KUKA KRL program: MyProgram_319().src

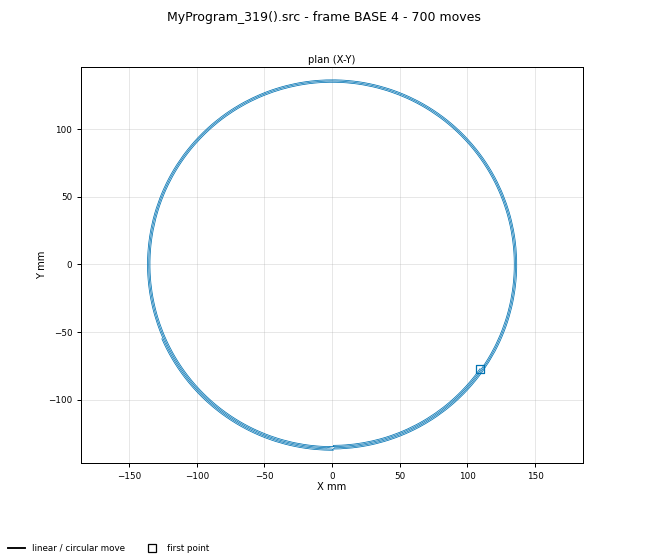
[picture p0: tool path of MyProgram_319().src in frame BASE 4, 700 of 700 moves have a stored position in this frame; points joined in program order, loops and branches not executed]
&ACCESS RVP
&REL 1
&PARAM TEMPLATE = C:\KRC\Roboter\Template\vorgabe
&PARAM EDITMASK = *
DEF MyProgram_319()
; ---- Setting reference (Base) ----
$BASE = BASE_DATA[4]

; --------------------------
; ---- Setting tool (TCP) ----
$TOOL = TOOL_DATA[3]
; --------------------------

$VEL.CP = VEL_APROX_PRINT
Startdeposition()
$VEL.CP = VEL_PRINT
LIN {X 109.3778,Y -77.0106,Z 185,A -30.8894,B 3.0839,C 0.2483,E1 3.2253,E2 483.8317} C_DIS
LIN {X 107.5202,Y -79.5843,Z 185,A -32.1533,B 3.0837,C 0.2506,E1 3.2233,E2 485.0845} C_DIS
LIN {X 105.6235,Y -82.0842,Z 185,A -33.5327,B 3.0834,C 0.2541,E1 3.2209,E2 486.4695} C_DIS
LIN {X 103.4321,Y -84.829,Z 185,A -34.958,B 3.0832,C 0.2567,E1 3.2184,E2 487.886} C_DIS
LIN {X 100.7853,Y -87.957,Z 185,A -36.6496,B 3.0829,C 0.26,E1 3.2154,E2 489.5709} C_DIS
LIN {X 98.5631,Y -90.4402,Z 185,A -38.0166,B 3.0827,C 0.2625,E1 3.2128,E2 490.9313} C_DIS
LIN {X 95.7665,Y -93.3971,Z 185,A -39.7017,B 3.0825,C 0.2657,E1 3.2096,E2 492.6104} C_DIS
LIN {X 93.4185,Y -95.7456,Z 185,A -41.0913,B 3.0822,C 0.2683,E1 3.2068,E2 493.997} C_DIS
LIN {X 90.4442,Y -98.5594,Z 185,A -42.9213,B 3.0819,C 0.2726,E1 3.203,E2 495.8381} C_DIS
LIN {X 87.3741,Y -101.2911,Z 185,A -44.4719,B 3.0817,C 0.2741,E1 3.1998,E2 497.3634} C_DIS
LIN {X 84.3456,Y -103.8272,Z 185,A -46.1519,B 3.0814,C 0.2772,E1 3.1962,E2 499.0432} C_DIS
LIN {X 81.6511,Y -105.9592,Z 185,A -47.6942,B 3.0811,C 0.2805,E1 3.1928,E2 500.5957} C_DIS
LIN {X 78.452,Y -108.3485,Z 185,A -49.2173,B 3.0811,C 0.2819,E1 3.1894,E2 502.0961} C_DIS
LIN {X 76.0517,Y -110.0474,Z 185,A -50.5208,B 3.0808,C 0.2845,E1 3.1864,E2 503.4062} C_DIS
LIN {X 72.8711,Y -112.1781,Z 185,A -52.0108,B 3.0807,C 0.2859,E1 3.183,E2 504.8783} C_DIS
LIN {X 70.2032,Y -113.8671,Z 185,A -53.3655,B 3.0804,C 0.2881,E1 3.1798,E2 506.2343} C_DIS
LIN {X 67.5529,Y -115.459,Z 185,A -54.6759,B 3.0803,C 0.2901,E1 3.1766,E2 507.5439} C_DIS
LIN {X 64.5814,Y -117.147,Z 185,A -56.059,B 3.0801,C 0.2916,E1 3.1733,E2 508.9177} C_DIS
LIN {X 61.6787,Y -118.6998,Z 185,A -57.4546,B 3.0799,C 0.2935,E1 3.1698,E2 510.3125} C_DIS
LIN {X 58.6673,Y -120.2166,Z 185,A -58.8657,B 3.0798,C 0.2952,E1 3.1663,E2 511.7203} C_DIS
LIN {X 55.7023,Y -121.6185,Z 185,A -60.239,B 3.0796,C 0.2968,E1 3.1628,E2 513.0906} C_DIS
LIN {X 53.1765,Y -122.743,Z 185,A -61.4788,B 3.0794,C 0.2988,E1 3.1596,E2 514.3383} C_DIS
LIN {X 49.6723,Y -124.203,Z 185,A -62.991,B 3.0794,C 0.2998,E1 3.1558,E2 515.837} C_DIS
LIN {X 46.6127,Y -125.3832,Z 185,A -64.3692,B 3.0792,C 0.3012,E1 3.1522,E2 517.2128} C_DIS
LIN {X 43.5231,Y -126.4889,Z 185,A -65.8758,B 3.079,C 0.3035,E1 3.1481,E2 518.7333} C_DIS
LIN {X 39.4666,Y -127.8128,Z 185,A -67.6587,B 3.0788,C 0.305,E1 3.1434,E2 520.5116} C_DIS
LIN {X 35.6745,Y -128.9228,Z 185,A -69.2121,B 3.0788,C 0.3055,E1 3.1393,E2 522.0482} C_DIS
LIN {X 32.5911,Y -129.7365,Z 185,A -70.5581,B 3.0787,C 0.3065,E1 3.1356,E2 523.3925} C_DIS
LIN {X 29.3997,Y -130.497,Z 185,A -71.9433,B 3.0786,C 0.3075,E1 3.1319,E2 524.776} C_DIS
LIN {X 26.191,Y -131.179,Z 185,A -73.3307,B 3.0785,C 0.3084,E1 3.1281,E2 526.162} C_DIS
LIN {X 22.9498,Y -131.7853,Z 185,A -74.7231,B 3.0785,C 0.3091,E1 3.1242,E2 527.5527} C_DIS
LIN {X 19.6218,Y -132.3222,Z 185,A -76.1756,B 3.0783,C 0.3101,E1 3.1202,E2 529.0071} C_DIS
LIN {X 16.4658,Y -132.7515,Z 185,A -77.5281,B 3.0783,C 0.3107,E1 3.1165,E2 530.3588} C_DIS
LIN {X 13.2073,Y -133.1144,Z 185,A -78.924,B 3.0782,C 0.3113,E1 3.1126,E2 531.7544} C_DIS
LIN {X 9.919,Y -133.3992,Z 185,A -80.3167,B 3.0782,C 0.3117,E1 3.1087,E2 533.1452} C_DIS
LIN {X 6.649,Y -133.6021,Z 185,A -81.7182,B 3.0782,C 0.3121,E1 3.1048,E2 534.5471} C_DIS
LIN {X 3.2803,Y -133.7279,Z 185,A -83.13,B 3.0781,C 0.3123,E1 3.1009,E2 535.9555} C_DIS
LIN {X 0.9683,Y -133.7631,Z 185,A -83.8532,B 3.0783,C 0.3106,E1 3.0989,E2 536.6446} C_DIS
Enddeposition()
LIN {X 0.9683,Y -133.7631,Z 185,A -83.8532,B 3.0783,C 0.3106,E1 3.0989,E2 536.6446} C_DIS
Startdeposition()
$VEL.CP = VEL_PRINT
LIN {X 1.3005,Y -134.6625,Z 185,A -83.2219,B 3.0781,C 0.3087,E1 3.1005,E2 535.98} C_DIS
LIN {X 4.845,Y -134.581,Z 185,A -81.7788,B 3.0781,C 0.3087,E1 3.1045,E2 534.5448} C_DIS
LIN {X 8.4966,Y -134.3994,Z 185,A -79.9996,B 3.0784,C 0.3065,E1 3.1095,E2 532.7353} C_DIS
LIN {X 11.7944,Y -134.1508,Z 185,A -78.8459,B 3.0782,C 0.3079,E1 3.1127,E2 531.6142} C_DIS
LIN {X 15.0407,Y -133.8264,Z 185,A -77.5552,B 3.0782,C 0.3079,E1 3.1162,E2 530.3356} C_DIS
LIN {X 18.6503,Y -133.3703,Z 185,A -76.1047,B 3.0782,C 0.3079,E1 3.1202,E2 528.897} C_DIS
LIN {X 22.1894,Y -132.8267,Z 185,A -74.5857,B 3.0783,C 0.307,E1 3.1244,E2 527.3777} C_DIS
LIN {X 26.0809,Y -132.12,Z 185,A -72.6662,B 3.0786,C 0.304,E1 3.1298,E2 525.4261} C_DIS
LIN {X 29.5428,Y -131.3876,Z 185,A -71.3256,B 3.0786,C 0.3042,E1 3.1334,E2 524.1063} C_DIS
LIN {X 32.2356,Y -130.7541,Z 185,A -70.0345,B 3.0788,C 0.3023,E1 3.1369,E2 522.7994} C_DIS
LIN {X 36.5633,Y -129.6089,Z 185,A -68.2253,B 3.0788,C 0.3013,E1 3.1418,E2 521.0015} C_DIS
LIN {X 40.7406,Y -128.357,Z 185,A -66.4521,B 3.079,C 0.3002,E1 3.1465,E2 519.238} C_DIS
LIN {X 44.2028,Y -127.206,Z 185,A -64.9326,B 3.0791,C 0.2988,E1 3.1505,E2 517.7217} C_DIS
LIN {X 46.9299,Y -126.2257,Z 185,A -63.7404,B 3.0792,C 0.2978,E1 3.1536,E2 516.534} C_DIS
LIN {X 50.2109,Y -124.9564,Z 185,A -62.2458,B 3.0794,C 0.296,E1 3.1575,E2 515.0386} C_DIS
LIN {X 53.1011,Y -123.7563,Z 185,A -61.1043,B 3.0794,C 0.296,E1 3.1604,E2 513.9212} C_DIS
LIN {X 56.2881,Y -122.3394,Z 185,A -59.4911,B 3.0797,C 0.293,E1 3.1645,E2 512.2899} C_DIS
LIN {X 59.0636,Y -121.0249,Z 185,A -58.3182,B 3.0797,C 0.2923,E1 3.1675,E2 511.1336} C_DIS
LIN {X 61.3147,Y -119.899,Z 185,A -56.7975,B 3.0802,C 0.2869,E1 3.1714,E2 509.5532} C_DIS
LIN {X 64.7424,Y -118.0858,Z 185,A -54.7565,B 3.0808,C 0.2811,E1 3.1765,E2 507.4594} C_DIS
LIN {X 70.0164,Y -115.0374,Z 185,A -52.4587,B 3.0809,C 0.2796,E1 3.1819,E2 505.1985} C_DIS
LIN {X 74.0705,Y -112.4692,Z 185,A -50.9669,B 3.0808,C 0.2811,E1 3.1852,E2 503.7774} C_DIS
LIN {X 77.8025,Y -109.9208,Z 185,A -49.3001,B 3.0808,C 0.28,E1 3.189,E2 502.1425} C_DIS
LIN {X 80.2283,Y -108.163,Z 185,A -47.8599,B 3.0812,C 0.2763,E1 3.1923,E2 500.6798} C_DIS
LIN {X 83.5783,Y -105.5962,Z 185,A -46.1074,B 3.0815,C 0.2734,E1 3.1961,E2 498.9314} C_DIS
LIN {X 87.2434,Y -102.5882,Z 185,A -44.1341,B 3.0818,C 0.2699,E1 3.2004,E2 496.9623} C_DIS
LIN {X 90.1434,Y -100.0503,Z 185,A -42.5344,B 3.082,C 0.2671,E1 3.2037,E2 495.3666} C_DIS
LIN {X 93.2151,Y -97.1943,Z 185,A -40.8836,B 3.0822,C 0.2647,E1 3.207,E2 493.7317} C_DIS
LIN {X 95.5931,Y -94.8563,Z 185,A -39.3699,B 3.0826,C 0.2609,E1 3.21,E2 492.2046} C_DIS
LIN {X 98.923,Y -91.3788,Z 185,A -37.4393,B 3.0828,C 0.2576,E1 3.2137,E2 490.2876} C_DIS
LIN {X 101.7497,Y -88.2209,Z 185,A -35.6928,B 3.0831,C 0.2542,E1 3.2169,E2 488.5471} C_DIS
LIN {X 104.4542,Y -85.0008,Z 185,A -34.0949,B 3.0833,C 0.252,E1 3.2197,E2 486.9725} C_DIS
LIN {X 106.6925,Y -82.1744,Z 185,A -32.5098,B 3.0836,C 0.248,E1 3.2224,E2 485.3796} C_DIS
LIN {X 108.6611,Y -79.5523,Z 185,A -30.8322,B 3.0841,C 0.242,E1 3.2253,E2 483.6641} C_DIS
LIN {X 111.066,Y -76.1584,Z 185,A -29.6154,B 3.0841,C 0.2431,E1 3.2271,E2 482.5176} C_DIS
LIN {X 113.0218,Y -73.2246,Z 185,A -28.0863,B 3.0843,C 0.2392,E1 3.2295,E2 480.9836} C_DIS
LIN {X 115.26,Y -69.6483,Z 185,A -26.3569,B 3.0846,C 0.2355,E1 3.232,E2 479.2612} C_DIS
LIN {X 117.2876,Y -66.1772,Z 185,A -24.733,B 3.0849,C 0.232,E1 3.2342,E2 477.6471} C_DIS
LIN {X 119.9686,Y -61.178,Z 185,A -22.4785,B 3.0852,C 0.2275,E1 3.2371,E2 475.4111} C_DIS
LIN {X 121.2175,Y -58.6685,Z 185,A -21.3605,B 3.0854,C 0.2251,E1 3.2385,E2 474.3018} C_DIS
LIN {X 122.8229,Y -55.2252,Z 185,A -19.8019,B 3.0856,C 0.2215,E1 3.2403,E2 472.7493} C_DIS
LIN {X 124.0307,Y -52.4592,Z 185,A -17.9985,B 3.0862,C 0.213,E1 3.2424,E2 470.8781} C_DIS
LIN {X 125.7519,Y -48.1884,Z 185,A -16.895,B 3.086,C 0.2163,E1 3.2434,E2 469.8829} C_DIS
LIN {X 128.0015,Y -41.8498,Z 185,A -13.8002,B 3.0867,C 0.2063,E1 3.2463,E2 466.7565} C_DIS
LIN {X 129.0855,Y -38.373,Z 185,A -12.3343,B 3.0869,C 0.2029,E1 3.2474,E2 465.3} C_DIS
LIN {X 130.1567,Y -34.5617,Z 185,A -10.7069,B 3.0872,C 0.1989,E1 3.2486,E2 463.6785} C_DIS
LIN {X 131.193,Y -30.3949,Z 185,A -8.9585,B 3.0874,C 0.1946,E1 3.2497,E2 461.9389} C_DIS
LIN {X 132.1228,Y -26.067,Z 185,A -7.1333,B 3.0877,C 0.19,E1 3.2508,E2 460.1197} C_DIS
LIN {X 132.6923,Y -22.9915,Z 185,A -6.0049,B 3.0878,C 0.1883,E1 3.2513,E2 459.0161} C_DIS
LIN {X 133.1849,Y -19.9387,Z 185,A -4.5848,B 3.0881,C 0.1836,E1 3.2519,E2 457.5817} C_DIS
LIN {X 133.671,Y -16.3571,Z 185,A -3.3283,B 3.0882,C 0.1821,E1 3.2523,E2 456.3598} C_DIS
LIN {X 134.1332,Y -12.0009,Z 185,A -1.3386,B 3.0886,C 0.1756,E1 3.2529,E2 454.3529} C_DIS
LIN {X 134.4654,Y -7.404,Z 185,A 0.3285,B 3.0887,C 0.173,E1 3.2532,E2 452.7217} C_DIS
LIN {X 134.6142,Y -3.7919,Z 185,A 1.9096,B 3.089,C 0.1682,E1 3.2533,E2 451.1341} C_DIS
LIN {X 134.6685,Y 0.4022,Z 185,A 3.7111,B 3.0893,C 0.163,E1 3.2533,E2 449.3293} C_DIS
LIN {X 134.5759,Y 4.9748,Z 185,A 5.2913,B 3.0893,C 0.1611,E1 3.2533,E2 447.7938} C_DIS
LIN {X 134.4125,Y 8.2847,Z 185,A 6.6289,B 3.0895,C 0.1579,E1 3.2531,E2 446.4644} C_DIS
LIN {X 134.1339,Y 11.9947,Z 185,A 8.4307,B 3.0899,C 0.1513,E1 3.2526,E2 444.6343} C_DIS
LIN {X 133.7255,Y 15.9002,Z 185,A 9.8128,B 3.0899,C 0.1494,E1 3.2522,E2 443.2873} C_DIS
LIN {X 133.4042,Y 18.4128,Z 185,A 10.8534,B 3.0901,C 0.1468,E1 3.2518,E2 442.2507} C_DIS
LIN {X 132.9214,Y 21.622,Z 185,A 12.337,B 3.0903,C 0.1419,E1 3.2512,E2 440.7535} C_DIS
LIN {X 132.3451,Y 24.9042,Z 185,A 13.6153,B 3.0904,C 0.1394,E1 3.2505,E2 439.4918} C_DIS
LIN {X 131.6524,Y 28.3359,Z 185,A 15.0387,B 3.0906,C 0.1359,E1 3.2497,E2 438.0758} C_DIS
LIN {X 130.8725,Y 31.7442,Z 185,A 16.4839,B 3.0907,C 0.1322,E1 3.2488,E2 436.6352} C_DIS
LIN {X 129.7931,Y 35.9048,Z 185,A 18.0917,B 3.0909,C 0.1294,E1 3.2477,E2 435.0538} C_DIS
LIN {X 128.8457,Y 39.1676,Z 185,A 19.6946,B 3.0911,C 0.1239,E1 3.2464,E2 433.4307} C_DIS
LIN {X 127.6225,Y 42.9879,Z 185,A 21.1611,B 3.0911,C 0.1217,E1 3.2451,E2 431.9932} C_DIS
LIN {X 126.451,Y 46.3233,Z 185,A 22.6096,B 3.0913,C 0.1182,E1 3.2438,E2 430.5509} C_DIS
LIN {X 124.7598,Y 50.6987,Z 185,A 24.7043,B 3.0915,C 0.112,E1 3.2416,E2 428.4432} C_DIS
LIN {X 123.3253,Y 54.098,Z 185,A 26.2489,B 3.0917,C 0.1082,E1 3.2399,E2 426.901} C_DIS
LIN {X 121.8233,Y 57.4005,Z 185,A 27.6922,B 3.0917,C 0.1051,E1 3.2382,E2 425.4696} C_DIS
LIN {X 120.1093,Y 60.9015,Z 185,A 29.1409,B 3.0919,C 0.1029,E1 3.2364,E2 424.0461} C_DIS
LIN {X 118.5408,Y 63.9051,Z 185,A 30.6264,B 3.0919,C 0.0989,E1 3.2345,E2 422.5547} C_DIS
LIN {X 116.1833,Y 68.0971,Z 185,A 32.5618,B 3.0921,C 0.0949,E1 3.2318,E2 420.6322} C_DIS
LIN {X 114.3594,Y 71.1174,Z 185,A 34.0309,B 3.0922,C 0.0915,E1 3.2297,E2 419.1666} C_DIS
LIN {X 111.9804,Y 74.8074,Z 185,A 35.7223,B 3.0922,C 0.0887,E1 3.2271,E2 417.4963} C_DIS
LIN {X 109.8113,Y 77.9576,Z 185,A 37.4338,B 3.0924,C 0.0841,E1 3.2243,E2 415.774} C_DIS
LIN {X 107.0698,Y 81.6813,Z 185,A 39.3105,B 3.0925,C 0.0804,E1 3.2212,E2 413.908} C_DIS
LIN {X 104.2356,Y 85.2683,Z 185,A 41.1787,B 3.0926,C 0.0768,E1 3.218,E2 412.0487} C_DIS
LIN {X 101.4876,Y 88.5213,Z 185,A 42.894,B 3.0926,C 0.0737,E1 3.2149,E2 410.3448} C_DIS
LIN {X 98.6491,Y 91.674,Z 185,A 44.6275,B 3.0928,C 0.0705,E1 3.2116,E2 408.6197} C_DIS
LIN {X 95.4237,Y 95.0268,Z 185,A 46.527,B 3.0928,C 0.0671,E1 3.2079,E2 406.7296} C_DIS
LIN {X 92.7076,Y 97.6791,Z 185,A 47.908,B 3.0928,C 0.0659,E1 3.2052,E2 405.3768} C_DIS
LIN {X 89.4844,Y 100.6402,Z 185,A 49.9683,B 3.093,C 0.0605,E1 3.2009,E2 403.2923} C_DIS
LIN {X 86.1879,Y 103.4773,Z 185,A 51.7785,B 3.093,C 0.0574,E1 3.197,E2 401.4868} C_DIS
LIN {X 82.5934,Y 106.3678,Z 185,A 53.6465,B 3.093,C 0.0546,E1 3.193,E2 399.6301} C_DIS
LIN {X 78.9904,Y 109.07,Z 185,A 55.5043,B 3.0931,C 0.0518,E1 3.1888,E2 397.7793} C_DIS
LIN {X 75.3567,Y 111.6116,Z 185,A 57.2001,B 3.0931,C 0.0502,E1 3.185,E2 396.1066} C_DIS
LIN {X 72.8837,Y 113.2423,Z 185,A 58.6152,B 3.0932,C 0.0469,E1 3.1816,E2 394.6729} C_DIS
LIN {X 68.9223,Y 115.6956,Z 185,A 60.5851,B 3.0932,C 0.0439,E1 3.1769,E2 392.7045} C_DIS
LIN {X 66.1927,Y 117.2789,Z 185,A 62.2054,B 3.0933,C 0.0397,E1 3.1729,E2 391.0508} C_DIS
LIN {X 62.5621,Y 119.2526,Z 185,A 63.5174,B 3.0933,C 0.0408,E1 3.1698,E2 389.7927} C_DIS
LIN {X 58.6336,Y 121.2342,Z 185,A 65.3547,B 3.0933,C 0.0386,E1 3.1652,E2 387.9598} C_DIS
LIN {X 55.3435,Y 122.77,Z 185,A 66.8326,B 3.0933,C 0.0371,E1 3.1614,E2 386.4901} C_DIS
LIN {X 52.0205,Y 124.2139,Z 185,A 68.2284,B 3.0933,C 0.0364,E1 3.1579,E2 385.1119} C_DIS
LIN {X 49.4921,Y 125.245,Z 185,A 69.4047,B 3.0933,C 0.035,E1 3.1548,E2 383.9342} C_DIS
LIN {X 45.9018,Y 126.603,Z 185,A 70.8196,B 3.0933,C 0.0349,E1 3.1512,E2 382.5455} C_DIS
LIN {X 42.9524,Y 127.6343,Z 185,A 72.3937,B 3.0933,C 0.0316,E1 3.1469,E2 380.9425} C_DIS
LIN {X 40.0856,Y 128.5647,Z 185,A 73.6526,B 3.0934,C 0.0306,E1 3.1436,E2 379.6868} C_DIS
LIN {X 36.8191,Y 129.5374,Z 185,A 74.9534,B 3.0934,C 0.0304,E1 3.1402,E2 378.4041} C_DIS
LIN {X 34.0373,Y 130.2966,Z 185,A 76.4081,B 3.0934,C 0.0277,E1 3.1361,E2 376.9226} C_DIS
LIN {X 29.8934,Y 131.3075,Z 185,A 78.0827,B 3.0934,C 0.0273,E1 3.1316,E2 375.2651} C_DIS
LIN {X 25.6894,Y 132.195,Z 185,A 79.8704,B 3.0934,C 0.0264,E1 3.1268,E2 373.4828} C_DIS
LIN {X 22.9962,Y 132.6914,Z 185,A 81.0398,B 3.0934,C 0.0257,E1 3.1235,E2 372.3133} C_DIS
LIN {X 19.0964,Y 133.3066,Z 185,A 82.6366,B 3.0934,C 0.0253,E1 3.1191,E2 370.7268} C_DIS
LIN {X 15.9212,Y 133.723,Z 185,A 84.042,B 3.0934,C 0.0244,E1 3.1152,E2 369.3168} C_DIS
LIN {X 10.8551,Y 134.2302,Z 185,A 86.3159,B 3.0934,C 0.0228,E1 3.1089,E2 367.0309} C_DIS
LIN {X 6.5583,Y 134.5079,Z 185,A 87.9984,B 3.0934,C 0.0233,E1 3.1042,E2 365.3669} C_DIS
LIN {X 2.4698,Y 134.6452,Z 185,A 89.6861,B 3.0934,C 0.0233,E1 3.0995,E2 363.6862} C_DIS
LIN {X -1.7718,Y 134.6568,Z 185,A 91.6474,B 3.0934,C 0.0221,E1 3.094,E2 361.707} C_DIS
LIN {X -6.1824,Y 134.5268,Z 185,A 93.4013,B 3.0934,C 0.0229,E1 3.0891,E2 359.9686} C_DIS
LIN {X -9.7803,Y 134.3119,Z 185,A 95.0179,B 3.0934,C 0.0225,E1 3.0846,E2 358.3429} C_DIS
LIN {X -13.1416,Y 134.025,Z 185,A 96.7108,B 3.0934,C 0.021,E1 3.0798,E2 356.6199} C_DIS
LIN {X -16.6086,Y 133.641,Z 185,A 97.9208,B 3.0934,C 0.0231,E1 3.0765,E2 355.4434} C_DIS
LIN {X -20.7882,Y 133.0533,Z 185,A 99.7684,B 3.0934,C 0.0233,E1 3.0714,E2 353.5905} C_DIS
LIN {X -24.7898,Y 132.367,Z 185,A 101.2894,B 3.0934,C 0.0252,E1 3.0673,E2 352.095} C_DIS
LIN {X -28.19,Y 131.6839,Z 185,A 102.9182,B 3.0934,C 0.0249,E1 3.0628,E2 350.4487} C_DIS
LIN {X -31.2799,Y 130.9844,Z 185,A 104.2927,B 3.0934,C 0.0255,E1 3.059,E2 349.0719} C_DIS
LIN {X -34.3154,Y 130.2224,Z 185,A 105.6447,B 3.0934,C 0.0262,E1 3.0554,E2 347.7181} C_DIS
LIN {X -37.2356,Y 129.4185,Z 185,A 106.8305,B 3.0934,C 0.0276,E1 3.0522,E2 346.5453} C_DIS
LIN {X -43.4299,Y 127.4739,Z 185,A 109.7036,B 3.0934,C 0.0291,E1 3.0446,E2 343.6609} C_DIS
LIN {X -50.2513,Y 124.9402,Z 185,A 113.3227,B 3.0934,C 0.029,E1 3.0349,E2 339.9812} C_DIS
LIN {X -54.1812,Y 123.2893,Z 185,A 114.7924,B 3.0934,C 0.0327,E1 3.0313,E2 338.5539} C_DIS
LIN {X -57.5817,Y 121.7367,Z 185,A 116.3857,B 3.0934,C 0.0344,E1 3.0272,E2 336.9613} C_DIS
LIN {X -60.2196,Y 120.4546,Z 185,A 117.573,B 3.0934,C 0.0362,E1 3.0243,E2 335.782} C_DIS
LIN {X -63.739,Y 118.6301,Z 185,A 119.3603,B 3.0934,C 0.0377,E1 3.0198,E2 333.9839} C_DIS
LIN {X -67.3996,Y 116.5892,Z 185,A 121.0325,B 3.0933,C 0.0406,E1 3.0158,E2 332.3261} C_DIS
LIN {X -69.5142,Y 115.3411,Z 185,A 122.2958,B 3.0933,C 0.0409,E1 3.0127,E2 331.0375} C_DIS
LIN {X -73.1954,Y 113.0407,Z 185,A 124.0125,B 3.0933,C 0.0442,E1 3.0087,E2 329.3376} C_DIS
LIN {X -77.9354,Y 109.827,Z 185,A 126.4287,B 3.0932,C 0.048,E1 3.0032,E2 326.9257} C_DIS
LIN {X -81.6351,Y 107.1048,Z 185,A 128.9192,B 3.0932,C 0.0486,E1 2.9974,E2 324.3724} C_DIS
LIN {X -84.266,Y 105.0479,Z 185,A 130.6008,B 3.0932,C 0.0498,E1 2.9937,E2 322.6604} C_DIS
LIN {X -87.6759,Y 102.2192,Z 185,A 132.1235,B 3.0931,C 0.0548,E1 2.9906,E2 321.1827} C_DIS
LIN {X -90.9693,Y 99.2994,Z 185,A 134.033,B 3.0931,C 0.058,E1 2.9866,E2 319.2702} C_DIS
LIN {X -94.0366,Y 96.4002,Z 185,A 136.4477,B 3.0931,C 0.0587,E1 2.9816,E2 316.7821} C_DIS
LIN {X -97.5607,Y 92.8315,Z 185,A 138.1008,B 3.0929,C 0.065,E1 2.9785,E2 315.1888} C_DIS
LIN {X -101.897,Y 88.0494,Z 185,A 140.9062,B 3.0928,C 0.0704,E1 2.9733,E2 312.3784} C_DIS
LIN {X -104.1498,Y 85.3733,Z 185,A 142.881,B 3.0928,C 0.0715,E1 2.9697,E2 310.3459} C_DIS
LIN {X -106.7805,Y 82.0595,Z 185,A 144.33,B 3.0926,C 0.0769,E1 2.9673,E2 308.9409} C_DIS
LIN {X -109.1666,Y 78.8572,Z 185,A 146.0509,B 3.0926,C 0.0806,E1 2.9644,E2 307.2186} C_DIS
LIN {X -111.2378,Y 75.9081,Z 185,A 148.1813,B 3.0925,C 0.0818,E1 2.961,E2 305.0168} C_DIS
LIN {X -113.7502,Y 72.0882,Z 185,A 149.7378,B 3.0923,C 0.0879,E1 2.9587,E2 303.5092} C_DIS
LIN {X -115.6692,Y 68.9666,Z 185,A 151.3648,B 3.0923,C 0.0913,E1 2.9563,E2 301.8751} C_DIS
LIN {X -117.9428,Y 65.0025,Z 185,A 153.3002,B 3.0921,C 0.0961,E1 2.9537,E2 299.9423} C_DIS
LIN {X -119.8337,Y 61.4429,Z 185,A 155.0991,B 3.0919,C 0.1,E1 2.9514,E2 298.1345} C_DIS
LIN {X -121.2175,Y 58.6685,Z 185,A 156.3812,B 3.0919,C 0.1034,E1 2.9498,E2 296.8579} C_DIS
LIN {X -123.0277,Y 54.7672,Z 185,A 158.3716,B 3.0917,C 0.1075,E1 2.9475,E2 294.8492} C_DIS
LIN {X -124.2698,Y 51.8868,Z 185,A 159.796,B 3.0916,C 0.1106,E1 2.9459,E2 293.4149} C_DIS
LIN {X -125.6958,Y 48.3326,Z 185,A 161.4084,B 3.0914,C 0.1149,E1 2.9442,E2 291.8058} C_DIS
LIN {X -126.9735,Y 44.8735,Z 185,A 163.2798,B 3.0914,C 0.118,E1 2.9424,E2 289.8987} C_DIS
LIN {X -128.0253,Y 41.7781,Z 185,A 164.5893,B 3.0912,C 0.122,E1 2.9413,E2 288.6002} C_DIS
LIN {X -129.0998,Y 38.3243,Z 185,A 166.2275,B 3.091,C 0.1258,E1 2.94,E2 286.9509} C_DIS
LIN {X -130.338,Y 33.8801,Z 185,A 168.3537,B 3.0908,C 0.1305,E1 2.9384,E2 284.8061} C_DIS
LIN {X -132.2754,Y 25.2688,Z 185,A 172.1548,B 3.0904,C 0.1407,E1 2.9362,E2 281.0022} C_DIS
LIN {X -132.9366,Y 21.5308,Z 185,A 173.8703,B 3.0902,C 0.1448,E1 2.9354,E2 279.2755} C_DIS
LIN {X -133.5106,Y 17.6142,Z 185,A 175.6639,B 3.09,C 0.1491,E1 2.9347,E2 277.4694} C_DIS
LIN {X -133.929,Y 14.0869,Z 185,A 177.1885,B 3.0898,C 0.1533,E1 2.9342,E2 275.9443} C_DIS
LIN {X -134.2944,Y 10.0203,Z 185,A 179.047,B 3.0895,C 0.1578,E1 2.9338,E2 274.0719} C_DIS
LIN {X -134.5044,Y 6.628,Z 185,A -179.3967,B 3.0893,C 0.1614,E1 2.9335,E2 272.5029} C_DIS
LIN {X -134.6452,Y 2.4704,Z 185,A -177.5256,B 3.0891,C 0.1661,E1 2.9334,E2 270.6203} C_DIS
LIN {X -134.6525,Y -2.0298,Z 185,A -175.5842,B 3.0888,C 0.1714,E1 2.9334,E2 268.6768} C_DIS
LIN {X -134.5349,Y -6.0226,Z 185,A -173.72,B 3.0886,C 0.1756,E1 2.9336,E2 266.7933} C_DIS
LIN {X -134.3102,Y -9.803,Z 185,A -172.058,B 3.0883,C 0.1799,E1 2.9339,E2 265.1258} C_DIS
LIN {X -133.9376,Y -14.007,Z 185,A -170.3361,B 3.088,C 0.1852,E1 2.9344,E2 263.4143} C_DIS
LIN {X -133.5729,Y -17.1384,Z 185,A -168.9389,B 3.0878,C 0.1887,E1 2.9348,E2 262.0108} C_DIS
LIN {X -133.1031,Y -20.4665,Z 185,A -167.2679,B 3.0876,C 0.1918,E1 2.9355,E2 260.3104} C_DIS
LIN {X -132.3663,Y -24.7933,Z 185,A -165.332,B 3.0873,C 0.1967,E1 2.9365,E2 258.367} C_DIS
LIN {X -131.5867,Y -28.6406,Z 185,A -163.6563,B 3.087,C 0.2013,E1 2.9375,E2 256.6915} C_DIS
LIN {X -130.7814,Y -32.1221,Z 185,A -161.9961,B 3.0868,C 0.2049,E1 2.9385,E2 255.0146} C_DIS
LIN {X -129.9052,Y -35.504,Z 185,A -160.3221,B 3.0866,C 0.2082,E1 2.9398,E2 253.3175} C_DIS
LIN {X -128.8517,Y -39.148,Z 185,A -158.0964,B 3.0864,C 0.2102,E1 2.9417,E2 251.0148} C_DIS
LIN {X -127.2502,Y -44.0754,Z 185,A -156.6747,B 3.0858,C 0.2191,E1 2.9428,E2 249.6937} C_DIS
LIN {X -126.1315,Y -47.1814,Z 185,A -154.9853,B 3.0856,C 0.2216,E1 2.9445,E2 247.9689} C_DIS
LIN {X -124.9868,Y -50.1356,Z 185,A -153.5997,B 3.0854,C 0.225,E1 2.9459,E2 246.5791} C_DIS
LIN {X -123.7512,Y -53.113,Z 185,A -152.1319,B 3.0851,C 0.2281,E1 2.9475,E2 245.0996} C_DIS
LIN {X -122.0645,Y -56.8826,Z 185,A -150.245,B 3.0849,C 0.232,E1 2.9497,E2 243.1969} C_DIS
LIN {X -120.1711,Y -60.7802,Z 185,A -148.2335,B 3.0846,C 0.2359,E1 2.9523,E2 241.1648} C_DIS
LIN {X -117.8729,Y -65.1288,Z 185,A -146.455,B 3.0841,C 0.2423,E1 2.9546,E2 239.4271} C_DIS
LIN {X -116.0972,Y -68.2436,Z 185,A -144.5744,B 3.0839,C 0.2444,E1 2.9572,E2 237.5018} C_DIS
LIN {X -113.7996,Y -72.01,Z 185,A -142.5765,B 3.0836,C 0.2483,E1 2.9602,E2 235.489} C_DIS
LIN {X -111.2867,Y -75.8367,Z 185,A -140.528,B 3.0833,C 0.2523,E1 2.9634,E2 233.4281} C_DIS
LIN {X -108.9895,Y -79.1015,Z 185,A -138.9727,B 3.0829,C 0.2567,E1 2.9659,E2 231.8916} C_DIS
LIN {X -106.7369,Y -82.1166,Z 185,A -137.1287,B 3.0827,C 0.2591,E1 2.9691,E2 230.0168} C_DIS
LIN {X -103.9503,Y -85.6167,Z 185,A -135.1969,B 3.0824,C 0.263,E1 2.9725,E2 228.0818} C_DIS
LIN {X -101.7086,Y -88.268,Z 185,A -133.6142,B 3.0822,C 0.2655,E1 2.9754,E2 226.4858} C_DIS
LIN {X -98.201,Y -92.1544,Z 185,A -131.3838,B 3.0818,C 0.2699,E1 2.9796,E2 224.2554} C_DIS
LIN {X -95.2075,Y -95.2442,Z 185,A -129.5155,B 3.0815,C 0.2733,E1 2.9833,E2 222.3824} C_DIS
LIN {X -92.3345,Y -98.0311,Z 185,A -127.7181,B 3.0812,C 0.276,E1 2.9869,E2 220.573} C_DIS
LIN {X -89.1274,Y -100.9557,Z 185,A -125.8294,B 3.081,C 0.279,E1 2.9909,E2 218.6791} C_DIS
LIN {X -86.0313,Y -103.6069,Z 185,A -124.0102,B 3.0807,C 0.2816,E1 2.9948,E2 216.849} C_DIS
LIN {X -82.4746,Y -106.4598,Z 185,A -122.0233,B 3.0805,C 0.2845,E1 2.9992,E2 214.856} C_DIS
LIN {X -78.8911,Y -109.142,Z 185,A -120.0503,B 3.0802,C 0.2871,E1 3.0036,E2 212.8742} C_DIS
LIN {X -75.1288,Y -111.7658,Z 185,A -118.0513,B 3.08,C 0.2897,E1 3.0082,E2 210.8689} C_DIS
LIN {X -71.3635,Y -114.2063,Z 185,A -116.0734,B 3.0798,C 0.2919,E1 3.0129,E2 208.882} C_DIS
LIN {X -68.1188,Y -116.1705,Z 185,A -114.2679,B 3.0797,C 0.293,E1 3.0173,E2 207.0514} C_DIS
LIN {X -65.3369,Y -117.7576,Z 185,A -113.148,B 3.0794,C 0.296,E1 3.02,E2 205.9631} C_DIS
LIN {X -61.6734,Y -119.7164,Z 185,A -111.2564,B 3.0792,C 0.2974,E1 3.0247,E2 204.0551} C_DIS
LIN {X -58.6087,Y -121.2461,Z 185,A -109.9691,B 3.079,C 0.3,E1 3.0279,E2 202.7897} C_DIS
LIN {X -55.3581,Y -122.7634,Z 185,A -108.2834,B 3.079,C 0.3006,E1 3.0322,E2 201.0829} C_DIS
LIN {X -52.3537,Y -124.0748,Z 185,A -106.9834,B 3.0787,C 0.3025,E1 3.0355,E2 199.7951} C_DIS
LIN {X -49.4995,Y -125.2421,Z 185,A -105.5703,B 3.0787,C 0.3031,E1 3.0392,E2 198.3686} C_DIS
LIN {X -45.8163,Y -126.6338,Z 185,A -103.9077,B 3.0785,C 0.3045,E1 3.0436,E2 196.7072} C_DIS
LIN {X -42.795,Y -127.6867,Z 185,A -102.7033,B 3.0784,C 0.3065,E1 3.0467,E2 195.523} C_DIS
LIN {X -40.0514,Y -128.5752,Z 185,A -101.3286,B 3.0784,C 0.3065,E1 3.0504,E2 194.1288} C_DIS
LIN {X -36.3564,Y -129.6668,Z 185,A -99.5707,B 3.0784,C 0.3067,E1 3.0552,E2 192.3548} C_DIS
LIN {X -33.0955,Y -130.5372,Z 185,A -98.3021,B 3.0781,C 0.3086,E1 3.0586,E2 191.1077} C_DIS
LIN {X -30.1972,Y -131.2381,Z 185,A -96.9498,B 3.0781,C 0.3086,E1 3.0623,E2 189.7441} C_DIS
LIN {X -27.5134,Y -131.8285,Z 185,A -95.7649,B 3.0781,C 0.3091,E1 3.0655,E2 188.5568} C_DIS
LIN {X -23.9634,Y -132.5183,Z 185,A -94.134,B 3.0781,C 0.3091,E1 3.07,E2 186.9132} C_DIS
LIN {X -20.8385,Y -133.0455,Z 185,A -92.8194,B 3.0781,C 0.3096,E1 3.0737,E2 185.6026} C_DIS
LIN {X -16.9748,Y -133.5943,Z 185,A -90.8607,B 3.0782,C 0.3079,E1 3.0792,E2 183.6041} C_DIS
LIN {X -11.5421,Y -134.1721,Z 185,A -88.941,B 3.0779,C 0.311,E1 3.0844,E2 181.7366} C_DIS
LIN {X -8.4078,Y -134.4049,Z 185,A -87.6596,B 3.0779,C 0.3114,E1 3.088,E2 180.4619} C_DIS
LIN {X -4.5739,Y -134.5916,Z 185,A -85.6288,B 3.0782,C 0.3085,E1 3.0938,E2 178.3783} C_DIS
LIN {X 0.966,Y -134.6616,Z 185,A -84.2905,B 3.0774,C 0.3155,E1 3.0972,E2 177.1719} C_DIS
Enddeposition()
LIN {X 0.966,Y -134.6616,Z 185,A -84.2907,B 3.0774,C 0.3155,E1 3.0972,E2 177.1722} C_DIS
Startdeposition()
$VEL.CP = VEL_PRINT
LIN {X -3.8672,Y -135.5126,Z 185,A -86.1247,B 3.077,C 0.3159,E1 3.0916,E2 179.0112} C_DIS
LIN {X -8.5541,Y -135.2977,Z 185,A -88.1962,B 3.077,C 0.3165,E1 3.0858,E2 181.0951} C_DIS
LIN {X -12.9771,Y -134.9451,Z 185,A -90.8299,B 3.0764,C 0.3216,E1 3.0782,E2 183.8282} C_DIS
LIN {X -19.1145,Y -134.2133,Z 185,A -92.3279,B 3.0772,C 0.3135,E1 3.0744,E2 185.1821} C_DIS
LIN {X -21.8513,Y -133.7957,Z 185,A -93.8541,B 3.077,C 0.3156,E1 3.0701,E2 186.7555} C_DIS
LIN {X -25.9901,Y -133.054,Z 185,A -95.5371,B 3.0772,C 0.3144,E1 3.0655,E2 188.4268} C_DIS
LIN {X -28.9335,Y -132.4443,Z 185,A -96.87,B 3.0772,C 0.3142,E1 3.0618,E2 189.7683} C_DIS
LIN {X -33.1674,Y -131.4476,Z 185,A -98.7564,B 3.0772,C 0.3136,E1 3.0567,E2 191.6615} C_DIS
LIN {X -36.5717,Y -130.5413,Z 185,A -100.2182,B 3.0773,C 0.3126,E1 3.0527,E2 193.1202} C_DIS
LIN {X -40.3012,Y -129.4401,Z 185,A -101.8498,B 3.0775,C 0.3114,E1 3.0484,E2 194.7507} C_DIS
LIN {X -43.9255,Y -128.2548,Z 185,A -103.5962,B 3.0775,C 0.3111,E1 3.0437,E2 196.515} C_DIS
LIN {X -47.4215,Y -127.0028,Z 185,A -105.413,B 3.0775,C 0.3113,E1 3.0388,E2 198.3643} C_DIS
LIN {X -50.5787,Y -125.7787,Z 185,A -106.2635,B 3.0779,C 0.3065,E1 3.0368,E2 199.1395} C_DIS
LIN {X -54.1105,Y -124.3006,Z 185,A -108.1986,B 3.0779,C 0.3069,E1 3.0317,E2 201.1163} C_DIS
LIN {X -57.3797,Y -122.8264,Z 185,A -109.6599,B 3.0781,C 0.305,E1 3.028,E2 202.5708} C_DIS
LIN {X -60.1478,Y -121.4938,Z 185,A -111.0913,B 3.0781,C 0.3044,E1 3.0244,E2 204.0196} C_DIS
LIN {X -64.2093,Y -119.3992,Z 185,A -113.1172,B 3.0783,C 0.3026,E1 3.0194,E2 206.058} C_DIS
LIN {X -68.3248,Y -117.0931,Z 185,A -115.0237,B 3.0786,C 0.2997,E1 3.0147,E2 207.9534} C_DIS
LIN {X -71.39,Y -115.2499,Z 185,A -116.6674,B 3.0787,C 0.2984,E1 3.0108,E2 209.6143} C_DIS
LIN {X -74.5873,Y -113.2067,Z 185,A -118.3461,B 3.0789,C 0.2965,E1 3.0068,E2 211.3028} C_DIS
LIN {X -78.1924,Y -110.7473,Z 185,A -120.2617,B 3.0792,C 0.2941,E1 3.0024,E2 213.2276} C_DIS
LIN {X -81.9694,Y -107.9823,Z 185,A -122.2915,B 3.0794,C 0.2913,E1 2.9978,E2 215.264} C_DIS
LIN {X -85.5115,Y -105.1994,Z 185,A -124.2573,B 3.0797,C 0.2885,E1 2.9935,E2 217.2378} C_DIS
LIN {X -88.9875,Y -102.2755,Z 185,A -126.1907,B 3.08,C 0.2853,E1 2.9894,E2 219.1728} C_DIS
LIN {X -92.1813,Y -99.4067,Z 185,A -128.0842,B 3.0803,C 0.2824,E1 2.9855,E2 221.0762} C_DIS
LIN {X -95.8147,Y -95.9098,Z 185,A -130.2468,B 3.0806,C 0.2786,E1 2.9812,E2 223.2426} C_DIS
LIN {X -98.6097,Y -93.033,Z 185,A -132.3327,B 3.0807,C 0.2771,E1 2.9771,E2 225.3784} C_DIS
LIN {X -101.2141,Y -90.1933,Z 185,A -133.7098,B 3.0811,C 0.2727,E1 2.9745,E2 226.7231} C_DIS
LIN {X -103.9974,Y -86.9689,Z 185,A -135.5605,B 3.0814,C 0.2692,E1 2.9712,E2 228.5798} C_DIS
LIN {X -106.865,Y -83.421,Z 185,A -137.5998,B 3.0817,C 0.2656,E1 2.9676,E2 230.633} C_DIS
LIN {X -109.3421,Y -80.1457,Z 185,A -139.3451,B 3.0821,C 0.2618,E1 2.9647,E2 232.379} C_DIS
LIN {X -111.9454,Y -76.4678,Z 185,A -141.3595,B 3.0824,C 0.258,E1 2.9615,E2 234.407} C_DIS
LIN {X -114.429,Y -72.6993,Z 185,A -143.3589,B 3.0827,C 0.254,E1 2.9584,E2 236.4175} C_DIS
LIN {X -116.781,Y -68.8569,Z 185,A -145.5669,B 3.083,C 0.2508,E1 2.9552,E2 238.6635} C_DIS
LIN {X -118.5241,Y -65.8107,Z 185,A -146.6353,B 3.0834,C 0.2455,E1 2.9538,E2 239.6786} C_DIS
LIN {X -119.6628,Y -63.7169,Z 185,A -147.9985,B 3.0834,C 0.2445,E1 2.952,E2 241.0868} C_DIS
LIN {X -121.4779,Y -60.1801,Z 185,A -149.6076,B 3.0838,C 0.2401,E1 2.9499,E2 242.6861} C_DIS
LIN {X -123.1978,Y -56.5763,Z 185,A -151.3099,B 3.0842,C 0.2359,E1 2.9479,E2 244.3897} C_DIS
LIN {X -124.5918,Y -53.4369,Z 185,A -152.8477,B 3.0844,C 0.2325,E1 2.9462,E2 245.9378} C_DIS
LIN {X -125.8482,Y -50.4063,Z 185,A -154.2821,B 3.0847,C 0.2291,E1 2.9447,E2 247.3776} C_DIS
LIN {X -127.3955,Y -46.3578,Z 185,A -156.051,B 3.085,C 0.2241,E1 2.9429,E2 249.1378} C_DIS
LIN {X -128.9639,Y -41.7975,Z 185,A -158.5715,B 3.0853,C 0.2206,E1 2.9406,E2 251.7181} C_DIS
LIN {X -130.1923,Y -37.7966,Z 185,A -160.2137,B 3.0857,C 0.2154,E1 2.9393,E2 253.3436} C_DIS
LIN {X -131.1684,Y -34.2616,Z 185,A -161.8667,B 3.0859,C 0.2116,E1 2.9381,E2 255.0087} C_DIS
LIN {X -132.1428,Y -30.2789,Z 185,A -163.6169,B 3.0862,C 0.2069,E1 2.937,E2 256.7602} C_DIS
LIN {X -132.8838,Y -26.8415,Z 185,A -165.1879,B 3.0865,C 0.2031,E1 2.9361,E2 258.341} C_DIS
LIN {X -133.5121,Y -23.5206,Z 185,A -166.6289,B 3.0867,C 0.1992,E1 2.9354,E2 259.7828} C_DIS
LIN {X -134.0251,Y -20.3951,Z 185,A -168.1198,B 3.0869,C 0.1961,E1 2.9347,E2 261.292} C_DIS
LIN {X -134.5986,Y -16.1802,Z 185,A -169.9835,B 3.0872,C 0.1913,E1 2.934,E2 263.1628} C_DIS
LIN {X -134.9865,Y -12.5458,Z 185,A -171.6109,B 3.0875,C 0.1873,E1 2.9336,E2 264.7997} C_DIS
LIN {X -135.3065,Y -8.4124,Z 185,A -173.4002,B 3.0878,C 0.1825,E1 2.9332,E2 266.5925} C_DIS
LIN {X -135.4773,Y -4.9607,Z 185,A -175.0695,B 3.088,C 0.1791,E1 2.933,E2 268.2868} C_DIS
LIN {X -135.568,Y -0.5102,Z 185,A -176.9414,B 3.0883,C 0.1738,E1 2.933,E2 270.1564} C_DIS
LIN {X -135.5194,Y 3.6242,Z 185,A -178.7898,B 3.0885,C 0.1692,E1 2.933,E2 272.0161} C_DIS
LIN {X -135.3581,Y 7.5741,Z 185,A 179.3635,B 3.0887,C 0.1652,E1 2.9333,E2 273.8835} C_DIS
LIN {X -135.0718,Y 11.5865,Z 185,A 177.7366,B 3.089,C 0.1601,E1 2.9337,E2 275.5002} C_DIS
LIN {X -134.7819,Y 14.5751,Z 185,A 176.3164,B 3.0892,C 0.1571,E1 2.9341,E2 276.9381} C_DIS
LIN {X -134.2373,Y 18.9462,Z 185,A 174.4025,B 3.0894,C 0.1521,E1 2.9348,E2 278.8572} C_DIS
LIN {X -133.6821,Y 22.5323,Z 185,A 172.8244,B 3.0896,C 0.148,E1 2.9355,E2 280.4397} C_DIS
LIN {X -133.0426,Y 26.0494,Z 185,A 171.1012,B 3.0898,C 0.1445,E1 2.9364,E2 282.1879} C_DIS
LIN {X -131.6881,Y 32.2022,Z 185,A 168.4661,B 3.0901,C 0.1371,E1 2.938,E2 284.8176} C_DIS
LIN {X -130.7655,Y 35.77,Z 185,A 166.1607,B 3.0901,C 0.1356,E1 2.9398,E2 287.213} C_DIS
LIN {X -129.3641,Y 40.546,Z 185,A 164.6528,B 3.0905,C 0.1278,E1 2.9409,E2 288.647} C_DIS
LIN {X -127.5156,Y 46.0246,Z 185,A 162.2887,B 3.0908,C 0.121,E1 2.9431,E2 290.9995} C_DIS
LIN {X -126.5536,Y 48.6104,Z 185,A 160.7889,B 3.0908,C 0.1192,E1 2.9446,E2 292.5392} C_DIS
LIN {X -125.1833,Y 52.0354,Z 185,A 159.2436,B 3.091,C 0.1151,E1 2.9462,E2 294.0816} C_DIS
LIN {X -122.6334,Y 57.7929,Z 185,A 156.4782,B 3.0912,C 0.1087,E1 2.9494,E2 296.8578} C_DIS
LIN {X -121.4433,Y 60.2502,Z 185,A 155.1841,B 3.0913,C 0.1063,E1 2.951,E2 298.1679} C_DIS
LIN {X -119.8493,Y 63.3621,Z 185,A 153.6662,B 3.0914,C 0.1028,E1 2.953,E2 299.6896} C_DIS
LIN {X -117.8201,Y 67.0631,Z 185,A 151.7381,B 3.0916,C 0.099,E1 2.9556,E2 301.6338} C_DIS
LIN {X -115.5968,Y 70.8265,Z 185,A 149.8425,B 3.0917,C 0.0947,E1 2.9583,E2 303.5339} C_DIS
LIN {X -113.2285,Y 74.5541,Z 185,A 147.0749,B 3.0917,C 0.0939,E1 2.9628,E2 306.4077} C_DIS
LIN {X -109.7194,Y 79.6284,Z 185,A 145.6136,B 3.092,C 0.0835,E1 2.9649,E2 307.7299} C_DIS
LIN {X -106.522,Y 83.8574,Z 185,A 142.4439,B 3.092,C 0.0823,E1 2.9705,E2 311.0094} C_DIS
LIN {X -103.9211,Y 87.0599,Z 185,A 140.4955,B 3.0921,C 0.0795,E1 2.974,E2 312.9807} C_DIS
LIN {X -100.7281,Y 90.7359,Z 185,A 138.9775,B 3.0923,C 0.073,E1 2.9767,E2 314.4329} C_DIS
LIN {X -98.0768,Y 93.5947,Z 185,A 136.9612,B 3.0923,C 0.0713,E1 2.9806,E2 316.4919} C_DIS
LIN {X -95.784,Y 95.9393,Z 185,A 135.7939,B 3.0924,C 0.0676,E1 2.9829,E2 317.6322} C_DIS
LIN {X -92.7271,Y 98.8983,Z 185,A 133.8905,B 3.0924,C 0.0647,E1 2.9868,E2 319.5468} C_DIS
LIN {X -89.4552,Y 101.8673,Z 185,A 131.9336,B 3.0925,C 0.0617,E1 2.9908,E2 321.513} C_DIS
LIN {X -85.9996,Y 104.8006,Z 185,A 130.0663,B 3.0926,C 0.0582,E1 2.9948,E2 323.3732} C_DIS
LIN {X -79.919,Y 109.5086,Z 185,A 126.6416,B 3.0926,C 0.0537,E1 3.0025,E2 326.8163} C_DIS
LIN {X -76.2926,Y 112.0651,Z 185,A 124.3861,B 3.0927,C 0.0526,E1 3.0078,E2 329.1155} C_DIS
LIN {X -73.016,Y 114.2264,Z 185,A 122.9681,B 3.0927,C 0.0491,E1 3.011,E2 330.5039} C_DIS
LIN {X -69.3657,Y 116.4793,Z 185,A 121.16,B 3.0928,C 0.0466,E1 3.0154,E2 332.3101} C_DIS
LIN {X -65.3293,Y 118.7908,Z 185,A 118.6215,B 3.0928,C 0.0469,E1 3.0217,E2 334.9148} C_DIS
LIN {X -60.9652,Y 121.087,Z 185,A 117.1481,B 3.0928,C 0.0414,E1 3.0252,E2 336.3148} C_DIS
LIN {X -58.3298,Y 122.3769,Z 185,A 115.8036,B 3.0928,C 0.0405,E1 3.0286,E2 337.6709} C_DIS
LIN {X -54.3528,Y 124.1959,Z 185,A 113.8657,B 3.0929,C 0.039,E1 3.0336,E2 339.6182} C_DIS
LIN {X -50.447,Y 125.8318,Z 185,A 111.5427,B 3.0929,C 0.0402,E1 3.0398,E2 342.0028} C_DIS
LIN {X -45.816,Y 127.5908,Z 185,A 110.0389,B 3.0929,C 0.0352,E1 3.0435,E2 343.436} C_DIS
LIN {X -42.3231,Y 128.7926,Z 185,A 108.2571,B 3.0929,C 0.0352,E1 3.0483,E2 345.2429} C_DIS
LIN {X -37.9167,Y 130.1571,Z 185,A 106.5348,B 3.0929,C 0.0325,E1 3.0529,E2 346.9372} C_DIS
LIN {X -34.8301,Y 131.0168,Z 185,A 105.0643,B 3.0929,C 0.0323,E1 3.0569,E2 348.4207} C_DIS
LIN {X -30.4466,Y 132.1045,Z 185,A 103.1406,B 3.0929,C 0.0314,E1 3.0621,E2 350.3451} C_DIS
LIN {X -27.0061,Y 132.8504,Z 185,A 101.7026,B 3.093,C 0.0304,E1 3.066,E2 351.7764} C_DIS
LIN {X -23.6792,Y 133.4837,Z 185,A 100.3083,B 3.093,C 0.0296,E1 3.0698,E2 353.1655} C_DIS
LIN {X -20.3887,Y 134.0261,Z 185,A 98.794,B 3.093,C 0.0298,E1 3.0741,E2 354.6916} C_DIS
LIN {X -16.1135,Y 134.6066,Z 185,A 96.6091,B 3.093,C 0.0316,E1 3.0802,E2 356.918} C_DIS
LIN {X -12.1852,Y 135.0211,Z 185,A 95.3417,B 3.093,C 0.0288,E1 3.0836,E2 358.1374} C_DIS
LIN {X -8.7728,Y 135.2843,Z 185,A 93.7692,B 3.093,C 0.0295,E1 3.088,E2 359.7241} C_DIS
LIN {X -4.2494,Y 135.502,Z 185,A 91.5442,B 3.093,C 0.0315,E1 3.0944,E2 361.9848} C_DIS
LIN {X -0.2958,Y 135.5682,Z 185,A 90.0416,B 3.093,C 0.0306,E1 3.0985,E2 363.4669} C_DIS
LIN {X 3.6567,Y 135.5185,Z 185,A 88.5937,B 3.093,C 0.0295,E1 3.1025,E2 364.8878} C_DIS
LIN {X 7.8471,Y 135.3413,Z 185,A 86.7312,B 3.093,C 0.0305,E1 3.1077,E2 366.7603} C_DIS
LIN {X 15.3821,Y 134.6938,Z 185,A 83.7576,B 3.093,C 0.0302,E1 3.1159,E2 369.7065} C_DIS
LIN {X 18.9782,Y 134.2328,Z 185,A 82.1582,B 3.093,C 0.0314,E1 3.1204,E2 371.3132} C_DIS
LIN {X 22.8202,Y 133.6341,Z 185,A 80.5877,B 3.093,C 0.0319,E1 3.1247,E2 372.8746} C_DIS
LIN {X 25.7208,Y 133.1054,Z 185,A 79.2646,B 3.093,C 0.0332,E1 3.1283,E2 374.2065} C_DIS
LIN {X 30.1923,Y 132.1626,Z 185,A 77.3984,B 3.093,C 0.0341,E1 3.1334,E2 376.0644} C_DIS
LIN {X 33.4305,Y 131.3809,Z 185,A 76.0228,B 3.093,C 0.035,E1 3.1371,E2 377.4357} C_DIS
LIN {X 37.0724,Y 130.4013,Z 185,A 74.4611,B 3.093,C 0.0361,E1 3.1413,E2 378.9933} C_DIS
LIN {X 39.7769,Y 129.6006,Z 185,A 73.2867,B 3.093,C 0.0371,E1 3.1445,E2 380.1653} C_DIS
LIN {X 43.0022,Y 128.5665,Z 185,A 71.8495,B 3.093,C 0.0385,E1 3.1483,E2 381.6029} C_DIS
LIN {X 48.047,Y 126.7685,Z 185,A 69.3685,B 3.0929,C 0.0426,E1 3.1549,E2 384.1093} C_DIS
LIN {X 52.5177,Y 124.9818,Z 185,A 67.6645,B 3.0929,C 0.0425,E1 3.1592,E2 385.7737} C_DIS
LIN {X 55.6368,Y 123.6249,Z 185,A 66.2541,B 3.0929,C 0.044,E1 3.1628,E2 387.1806} C_DIS
LIN {X 58.6801,Y 122.2096,Z 185,A 64.8525,B 3.0929,C 0.0457,E1 3.1663,E2 388.5801} C_DIS
LIN {X 61.6345,Y 120.7463,Z 185,A 63.4535,B 3.0928,C 0.0477,E1 3.1698,E2 389.9796} C_DIS
LIN {X 65.0311,Y 118.9537,Z 185,A 61.8494,B 3.0928,C 0.0498,E1 3.1737,E2 391.5814} C_DIS
LIN {X 67.4861,Y 117.5788,Z 185,A 60.6193,B 3.0928,C 0.0519,E1 3.1767,E2 392.8162} C_DIS
LIN {X 71.3207,Y 115.2931,Z 185,A 58.8754,B 3.0927,C 0.0537,E1 3.1809,E2 394.5431} C_DIS
LIN {X 74.7997,Y 113.0669,Z 185,A 57.1334,B 3.0927,C 0.0565,E1 3.185,E2 396.2846} C_DIS
LIN {X 78.2397,Y 110.714,Z 185,A 55.3633,B 3.0926,C 0.0595,E1 3.189,E2 398.0557} C_DIS
LIN {X 82.0053,Y 107.9551,Z 185,A 53.471,B 3.0926,C 0.0623,E1 3.1932,E2 399.9385} C_DIS
LIN {X 85.4582,Y 105.243,Z 185,A 51.6529,B 3.0925,C 0.0654,E1 3.1972,E2 401.7522} C_DIS
LIN {X 88.7849,Y 102.4521,Z 185,A 49.8621,B 3.0924,C 0.0685,E1 3.201,E2 403.5378} C_DIS
LIN {X 94.6978,Y 97.0126,Z 185,A 46.7584,B 3.0924,C 0.0727,E1 3.2073,E2 406.6067} C_DIS
LIN {X 98.8254,Y 92.8044,Z 185,A 44.2659,B 3.0922,C 0.0779,E1 3.2121,E2 409.0998} C_DIS
LIN {X 101.4161,Y 89.9657,Z 185,A 42.6066,B 3.0921,C 0.0816,E1 3.2152,E2 410.7637} C_DIS
LIN {X 104.3069,Y 86.5974,Z 185,A 40.8023,B 3.092,C 0.0851,E1 3.2185,E2 412.5596} C_DIS
LIN {X 107.1251,Y 83.0856,Z 185,A 38.9747,B 3.0919,C 0.0887,E1 3.2216,E2 414.3786} C_DIS
LIN {X 109.9203,Y 79.3511,Z 185,A 37.0752,B 3.0918,C 0.0926,E1 3.2248,E2 416.2698} C_DIS
LIN {X 112.42,Y 75.7683,Z 185,A 35.2649,B 3.0916,C 0.0966,E1 3.2276,E2 418.0763} C_DIS
LIN {X 115.0184,Y 71.7621,Z 185,A 33.3306,B 3.0916,C 0.1007,E1 3.2305,E2 420.001} C_DIS
LIN {X 118.1353,Y 66.5061,Z 185,A 31.2387,B 3.0915,C 0.1025,E1 3.2334,E2 422.0337} C_DIS
LIN {X 120.1883,Y 62.7164,Z 185,A 29.205,B 3.0912,C 0.109,E1 3.2361,E2 424.094} C_DIS
LIN {X 122.0501,Y 59.0139,Z 185,A 27.2899,B 3.091,C 0.1151,E1 3.2385,E2 426.0298} C_DIS
LIN {X 124.0281,Y 54.7353,Z 185,A 25.6295,B 3.091,C 0.1171,E1 3.2403,E2 427.6504} C_DIS
LIN {X 125.3146,Y 51.7208,Z 185,A 24.1377,B 3.0908,C 0.1217,E1 3.242,E2 429.1558} C_DIS
LIN {X 127.284,Y 46.667,Z 185,A 22.1412,B 3.0906,C 0.1249,E1 3.2439,E2 431.1169} C_DIS
LIN {X 128.2266,Y 44.0069,Z 185,A 20.868,B 3.0905,C 0.1289,E1 3.2451,E2 432.4006} C_DIS
LIN {X 129.5498,Y 39.9429,Z 185,A 19.1828,B 3.0903,C 0.1326,E1 3.2465,E2 434.0717} C_DIS
LIN {X 130.5829,Y 36.423,Z 185,A 17.6951,B 3.0902,C 0.1362,E1 3.2476,E2 435.5524} C_DIS
LIN {X 131.475,Y 33.0595,Z 185,A 16.3038,B 3.09,C 0.1394,E1 3.2486,E2 436.9346} C_DIS
LIN {X 132.4573,Y 28.8736,Z 185,A 14.5405,B 3.0898,C 0.1439,E1 3.2497,E2 438.6922} C_DIS
LIN {X 133.257,Y 24.9278,Z 185,A 12.863,B 3.0896,C 0.1484,E1 3.2506,E2 440.3677} C_DIS
LIN {X 133.9602,Y 20.814,Z 185,A 11.2367,B 3.0894,C 0.152,E1 3.2513,E2 441.9778} C_DIS
LIN {X 134.5051,Y 16.9531,Z 185,A 9.4114,B 3.0891,C 0.1583,E1 3.252,E2 443.8262} C_DIS
LIN {X 134.8832,Y 13.6215,Z 185,A 8.4157,B 3.0891,C 0.1581,E1 3.2523,E2 444.7703} C_DIS
LIN {X 135.3778,Y 7.1828,Z 185,A 5.9117,B 3.0888,C 0.1636,E1 3.2528,E2 447.2479} C_DIS
LIN {X 135.5025,Y 4.2327,Z 185,A 3.9517,B 3.0883,C 0.1741,E1 3.253,E2 449.2975} C_DIS
LIN {X 135.5661,Y -0.8143,Z 185,A 2.3517,B 3.0883,C 0.1749,E1 3.253,E2 450.8325} C_DIS
LIN {X 135.4795,Y -4.9062,Z 185,A 0.8269,B 3.088,C 0.1778,E1 3.2528,E2 452.3327} C_DIS
LIN {X 135.2864,Y -8.7378,Z 185,A -0.6962,B 3.0878,C 0.1813,E1 3.2526,E2 453.8446} C_DIS
LIN {X 134.5275,Y -16.7766,Z 185,A -3.9167,B 3.0874,C 0.1891,E1 3.2517,E2 457.0433} C_DIS
LIN {X 134.1311,Y -19.6897,Z 185,A -5.0994,B 3.0872,C 0.1919,E1 3.2512,E2 458.2193} C_DIS
LIN {X 133.6307,Y -22.8406,Z 185,A -6.3926,B 3.087,C 0.1951,E1 3.2507,E2 459.5064} C_DIS
LIN {X 133.0072,Y -26.2348,Z 185,A -7.9545,B 3.0867,C 0.2002,E1 3.2498,E2 461.0825} C_DIS
LIN {X 132.1862,Y -30.0889,Z 185,A -9.4227,B 3.0865,C 0.2029,E1 3.249,E2 462.5269} C_DIS
LIN {X 131.3809,Y -33.4305,Z 185,A -10.8026,B 3.0863,C 0.2061,E1 3.248,E2 463.8987} C_DIS
LIN {X 130.5362,Y -36.5899,Z 185,A -12.1715,B 3.086,C 0.2098,E1 3.247,E2 465.2669} C_DIS
LIN {X 129.5629,Y -39.9,Z 185,A -13.5605,B 3.0858,C 0.2131,E1 3.2459,E2 466.6482} C_DIS
LIN {X 128.1189,Y -44.3176,Z 185,A -15.5999,B 3.0854,C 0.2191,E1 3.2441,E2 468.6987} C_DIS
LIN {X 126.7602,Y -48.0693,Z 185,A -17.1034,B 3.0852,C 0.2218,E1 3.2427,E2 470.1802} C_DIS
LIN {X 124.9957,Y -52.4845,Z 185,A -18.9441,B 3.0849,C 0.2255,E1 3.2407,E2 472.0009} C_DIS
LIN {X 123.4342,Y -56.0631,Z 185,A -20.5285,B 3.0847,C 0.2291,E1 3.239,E2 473.5783} C_DIS
LIN {X 122.1764,Y -58.7496,Z 185,A -21.7389,B 3.0845,C 0.2319,E1 3.2375,E2 474.7841} C_DIS
LIN {X 120.5244,Y -62.0704,Z 185,A -23.3835,B 3.0841,C 0.2367,E1 3.2354,E2 476.4399} C_DIS
LIN {X 117.0321,Y -68.4293,Z 185,A -26.2354,B 3.0837,C 0.2423,E1 3.2316,E2 479.2668} C_DIS
LIN {X 114.9506,Y -71.8711,Z 185,A -27.8777,B 3.0834,C 0.2459,E1 3.2292,E2 480.903} C_DIS
LIN {X 110.9375,Y -77.9228,Z 185,A -30.8235,B 3.0829,C 0.2521,E1 3.2246,E2 483.8356} C_DIS
LIN {X 109.125,Y -80.4413,Z 185,A -32.1254,B 3.0826,C 0.255,E1 3.2224,E2 485.1373} C_DIS
LIN {X 106.3599,Y -84.0639,Z 185,A -34.0689,B 3.0823,C 0.2596,E1 3.2191,E2 487.0845} C_DIS
LIN {X 103.4501,Y -87.6193,Z 185,A -35.813,B 3.082,C 0.2621,E1 3.216,E2 488.8047} C_DIS
LIN {X 100.0676,Y -91.4639,Z 185,A -37.9052,B 3.0817,C 0.2662,E1 3.2122,E2 490.8894} C_DIS
LIN {X 97.3358,Y -94.365,Z 185,A -39.9367,B 3.0811,C 0.2729,E1 3.2081,E2 492.967} C_DIS
LIN {X 94.3605,Y -97.3402,Z 185,A -41.1645,B 3.0812,C 0.2715,E1 3.2058,E2 494.1251} C_DIS
LIN {X 90.4196,Y -101.0114,Z 185,A -43.4644,B 3.0808,C 0.2763,E1 3.2011,E2 496.43} C_DIS
LIN {X 87.1877,Y -103.8139,Z 185,A -45.4903,B 3.0803,C 0.2817,E1 3.1967,E2 498.4855} C_DIS
LIN {X 84.4628,Y -106.0427,Z 185,A -46.4596,B 3.0805,C 0.2798,E1 3.1947,E2 499.3887} C_DIS
LIN {X 81.9712,Y -107.9809,Z 185,A -48.2562,B 3.0799,C 0.2864,E1 3.1906,E2 501.2464} C_DIS
LIN {X 79.0409,Y -110.1435,Z 185,A -49.4999,B 3.0799,C 0.2864,E1 3.1879,E2 502.453} C_DIS
LIN {X 75.5089,Y -112.5944,Z 185,A -51.2426,B 3.0796,C 0.2889,E1 3.1839,E2 504.1874} C_DIS
LIN {X 70.7535,Y -115.6416,Z 185,A -53.971,B 3.079,C 0.2958,E1 3.1773,E2 506.9619} C_DIS
LIN {X 67.022,Y -117.8431,Z 185,A -55.3084,B 3.0791,C 0.2943,E1 3.1742,E2 508.2365} C_DIS
LIN {X 63.6762,Y -119.6843,Z 185,A -56.9553,B 3.0789,C 0.2969,E1 3.1701,E2 509.8889} C_DIS
LIN {X 59.5855,Y -121.7711,Z 185,A -58.7361,B 3.0788,C 0.2983,E1 3.1657,E2 511.6502} C_DIS
LIN {X 56.1283,Y -123.405,Z 185,A -60.4245,B 3.0785,C 0.301,E1 3.1614,E2 513.3493} C_DIS
LIN {X 52.3885,Y -125.0358,Z 185,A -62.0138,B 3.0784,C 0.3021,E1 3.1574,E2 514.9221} C_DIS
LIN {X 48.9961,Y -126.4036,Z 185,A -63.5649,B 3.0782,C 0.3039,E1 3.1534,E2 516.4748} C_DIS
LIN {X 45.17,Y -127.8234,Z 185,A -65.4284,B 3.0779,C 0.307,E1 3.1484,E2 518.3577} C_DIS
LIN {X 41.8939,Y -128.9335,Z 185,A -66.7723,B 3.0779,C 0.3075,E1 3.1449,E2 519.6872} C_DIS
LIN {X 38.11,Y -130.1005,Z 185,A -68.322,B 3.0778,C 0.3081,E1 3.1408,E2 521.2217} C_DIS
LIN {X 34.6171,Y -131.0736,Z 185,A -69.825,B 3.0777,C 0.3093,E1 3.1367,E2 522.7218} C_DIS
LIN {X 30.7427,Y -132.0369,Z 185,A -71.5938,B 3.0775,C 0.3113,E1 3.1319,E2 524.5025} C_DIS
LIN {X 27.0638,Y -132.8386,Z 185,A -73.1008,B 3.0775,C 0.3118,E1 3.1278,E2 525.9992} C_DIS
LIN {X 21.4567,Y -133.8607,Z 185,A -75.3972,B 3.0773,C 0.3125,E1 3.1215,E2 528.2825} C_DIS
LIN {X 17.6878,Y -134.4088,Z 185,A -77.0245,B 3.0773,C 0.3135,E1 3.117,E2 529.9129} C_DIS
LIN {X 14.4061,Y -134.8001,Z 185,A -78.8392,B 3.0768,C 0.3173,E1 3.1118,E2 531.783} C_DIS
LIN {X 10.4163,Y -135.168,Z 185,A -80.2587,B 3.077,C 0.316,E1 3.1079,E2 533.1677} C_DIS
LIN {X 4.4954,Y -135.4952,Z 185,A -82.5561,B 3.077,C 0.3152,E1 3.1016,E2 535.4391} C_DIS
LIN {X 1.5859,Y -135.5602,Z 185,A -84.5418,B 3.0765,C 0.3209,E1 3.0958,E2 537.5238} C_DIS
LIN {X 1.5859,Y -135.5602,Z 185,A -84.5418,B 3.0765,C 0.3209,E1 3.0958,E2 537.5239} C_DIS
Enddeposition()
LIN {X 0.9629,Y -136.4645,Z 185,A -83.8807,B 3.1112,C 0.3172,E1 3.1321,E2 536.7633} C_DIS
Startdeposition()
$VEL.CP = VEL_PRINT
LIN {X 5.9779,Y -136.3384,Z 185,A -81.12,B 3.1117,C 0.3118,E1 3.14,E2 533.9146} C_DIS
LIN {X 15.0042,Y -135.6411,Z 185,A -77.647,B 3.1117,C 0.3127,E1 3.1496,E2 530.4835} C_DIS
LIN {X 17.9428,Y -135.2832,Z 185,A -76.0532,B 3.1119,C 0.3093,E1 3.1541,E2 528.8422} C_DIS
LIN {X 21.35,Y -134.7881,Z 185,A -74.6849,B 3.1119,C 0.3091,E1 3.1579,E2 527.4834} C_DIS
LIN {X 25.6706,Y -134.0315,Z 185,A -73.0876,B 3.1119,C 0.3098,E1 3.1622,E2 525.9176} C_DIS
LIN {X 28.7602,Y -133.4026,Z 185,A -71.7769,B 3.1119,C 0.3089,E1 3.1657,E2 524.6079} C_DIS
LIN {X 32.119,Y -132.6341,Z 185,A -70.3751,B 3.1121,C 0.3081,E1 3.1695,E2 523.2111} C_DIS
LIN {X 35.3624,Y -131.8065,Z 185,A -68.9905,B 3.1121,C 0.307,E1 3.1733,E2 521.8285} C_DIS
LIN {X 38.3015,Y -130.9824,Z 185,A -67.7204,B 3.1123,C 0.3059,E1 3.1767,E2 520.559} C_DIS
LIN {X 41.7371,Y -129.9286,Z 185,A -66.2,B 3.1124,C 0.3043,E1 3.1808,E2 519.036} C_DIS
LIN {X 46.5285,Y -128.2908,Z 185,A -64.1143,B 3.1126,C 0.3024,E1 3.1863,E2 516.9544} C_DIS
LIN {X 50.4958,Y -126.7827,Z 185,A -62.325,B 3.1128,C 0.3003,E1 3.1909,E2 515.1629} C_DIS
LIN {X 54.3036,Y -125.1978,Z 185,A -60.7733,B 3.1128,C 0.2997,E1 3.1949,E2 513.6339} C_DIS
LIN {X 57.3961,Y -123.8105,Z 185,A -59.2615,B 3.1131,C 0.297,E1 3.1987,E2 512.1093} C_DIS
LIN {X 60.7288,Y -122.2109,Z 185,A -57.7951,B 3.1133,C 0.2956,E1 3.2024,E2 510.6531} C_DIS
LIN {X 64.0124,Y -120.5245,Z 185,A -56.2906,B 3.1134,C 0.2938,E1 3.2061,E2 509.1536} C_DIS
LIN {X 69.1177,Y -117.6717,Z 185,A -53.69,B 3.1139,C 0.2888,E1 3.2125,E2 506.532} C_DIS
LIN {X 73.9114,Y -114.7221,Z 185,A -51.539,B 3.1141,C 0.2869,E1 3.2175,E2 504.4073} C_DIS
LIN {X 77.3633,Y -112.4226,Z 185,A -49.7937,B 3.1144,C 0.2839,E1 3.2215,E2 502.6602} C_DIS
LIN {X 83.4562,Y -107.9768,Z 185,A -46.2742,B 3.1152,C 0.275,E1 3.2295,E2 499.0914} C_DIS
LIN {X 87.0885,Y -105.069,Z 185,A -44.833,B 3.1151,C 0.2761,E1 3.2325,E2 497.7168} C_DIS
LIN {X 90.5053,Y -102.1406,Z 185,A -42.7226,B 3.1156,C 0.2703,E1 3.237,E2 495.5755} C_DIS
LIN {X 93.2449,Y -99.6463,Z 185,A -41.5741,B 3.1156,C 0.271,E1 3.2392,E2 494.4797} C_DIS
LIN {X 97.4295,Y -95.5582,Z 185,A -39.2107,B 3.1159,C 0.2668,E1 3.2439,E2 492.1267} C_DIS
LIN {X 100.0947,Y -92.7634,Z 185,A -37.4292,B 3.1163,C 0.2618,E1 3.2474,E2 490.3227} C_DIS
LIN {X 103.34,Y -89.1333,Z 185,A -35.5915,B 3.1165,C 0.2593,E1 3.2507,E2 488.5107} C_DIS
LIN {X 106.111,Y -85.816,Z 185,A -33.9663,B 3.1167,C 0.2571,E1 3.2535,E2 486.9089} C_DIS
LIN {X 108.3131,Y -83.0192,Z 185,A -32.3831,B 3.117,C 0.2528,E1 3.2563,E2 485.3128} C_DIS
LIN {X 110.8711,Y -79.571,Z 185,A -29.4056,B 3.1183,C 0.237,E1 3.2614,E2 482.178} C_DIS
LIN {X 115.9291,Y -72.0025,Z 185,A -27.1864,B 3.1178,C 0.2436,E1 3.2644,E2 480.168} C_DIS
LIN {X 120.4447,Y -64.1644,Z 185,A -23.4048,B 3.1185,C 0.2343,E1 3.2696,E2 476.3859} C_DIS
LIN {X 122.5741,Y -59.9926,Z 185,A -21.4824,B 3.1188,C 0.2297,E1 3.272,E2 474.4677} C_DIS
LIN {X 124.0018,Y -56.9825,Z 185,A -20.1634,B 3.119,C 0.2269,E1 3.2736,E2 473.1579} C_DIS
LIN {X 125.7109,Y -53.1078,Z 185,A -18.5587,B 3.1192,C 0.2239,E1 3.2753,E2 471.5744} C_DIS
LIN {X 127.3112,Y -49.146,Z 185,A -16.7053,B 3.1196,C 0.2186,E1 3.2772,E2 469.7119} C_DIS
LIN {X 128.5616,Y -45.7774,Z 185,A -14.9811,B 3.12,C 0.2124,E1 3.2789,E2 467.9584} C_DIS
LIN {X 129.6903,Y -42.4765,Z 185,A -13.9286,B 3.12,C 0.2126,E1 3.2798,E2 466.9585} C_DIS
LIN {X 130.9656,Y -38.359,Z 185,A -12.1317,B 3.1204,C 0.2078,E1 3.2812,E2 465.1618} C_DIS
LIN {X 131.9289,Y -34.9031,Z 185,A -10.7776,B 3.1205,C 0.2052,E1 3.2822,E2 463.8263} C_DIS
LIN {X 132.673,Y -31.9574,Z 185,A -9.4985,B 3.1208,C 0.2017,E1 3.2831,E2 462.5458} C_DIS
LIN {X 133.4146,Y -28.7049,Z 185,A -8.1392,B 3.121,C 0.1982,E1 3.2839,E2 461.1907} C_DIS
LIN {X 134.1758,Y -24.9158,Z 185,A -6.6113,B 3.1212,C 0.1947,E1 3.2847,E2 459.6739} C_DIS
LIN {X 134.7137,Y -21.8193,Z 185,A -5.3555,B 3.1214,C 0.1916,E1 3.2853,E2 458.4254} C_DIS
LIN {X 135.1491,Y -18.9291,Z 185,A -4.1237,B 3.1216,C 0.1882,E1 3.2858,E2 457.1921} C_DIS
LIN {X 135.8756,Y -12.7048,Z 185,A -1.4265,B 3.1221,C 0.1801,E1 3.2866,E2 454.4846} C_DIS
LIN {X 136.2343,Y -7.9915,Z 185,A 0.9899,B 3.1226,C 0.1701,E1 3.287,E2 452.011} C_DIS
LIN {X 136.4507,Y -2.1724,Z 185,A 2.743,B 3.1226,C 0.1703,E1 3.287,E2 450.3456} C_DIS
LIN {X 136.4122,Y 3.9021,Z 185,A 4.929,B 3.1228,C 0.1667,E1 3.287,E2 448.2046} C_DIS
LIN {X 135.9092,Y 12.3542,Z 185,A 8.3782,B 3.1233,C 0.1578,E1 3.2864,E2 444.767} C_DIS
LIN {X 135.2764,Y 17.9948,Z 185,A 10.6437,B 3.1236,C 0.1523,E1 3.2856,E2 442.5151} C_DIS
LIN {X 134.819,Y 21.1505,Z 185,A 12.0226,B 3.1238,C 0.1482,E1 3.2851,E2 441.1303} C_DIS
LIN {X 134.071,Y 25.4638,Z 185,A 13.783,B 3.124,C 0.1439,E1 3.2842,E2 439.3788} C_DIS
LIN {X 133.3272,Y 29.1096,Z 185,A 15.2366,B 3.1241,C 0.1406,E1 3.2834,E2 437.9381} C_DIS
LIN {X 132.6285,Y 32.1421,Z 185,A 16.511,B 3.1242,C 0.1374,E1 3.2825,E2 436.667} C_DIS
LIN {X 131.8266,Y 35.2867,Z 185,A 17.8188,B 3.1244,C 0.1342,E1 3.2816,E2 435.3654} C_DIS
LIN {X 130.8894,Y 38.6193,Z 185,A 19.1871,B 3.1245,C 0.1311,E1 3.2806,E2 434.0072} C_DIS
LIN {X 129.8539,Y 41.9709,Z 185,A 20.5572,B 3.1246,C 0.1281,E1 3.2794,E2 432.6493} C_DIS
LIN {X 128.9288,Y 44.7295,Z 185,A 21.8542,B 3.1248,C 0.1241,E1 3.2782,E2 431.3423} C_DIS
LIN {X 126.3366,Y 51.6007,Z 185,A 24.7125,B 3.125,C 0.1182,E1 3.2754,E2 428.5109} C_DIS
LIN {X 125.0689,Y 54.6018,Z 185,A 26.1086,B 3.1252,C 0.1143,E1 3.2739,E2 427.1107} C_DIS
LIN {X 123.6487,Y 57.746,Z 185,A 27.4481,B 3.1252,C 0.1117,E1 3.2723,E2 425.7843} C_DIS
LIN {X 122.2676,Y 60.614,Z 185,A 28.739,B 3.1254,C 0.1087,E1 3.2707,E2 424.4987} C_DIS
LIN {X 120.3957,Y 64.2567,Z 185,A 30.494,B 3.1255,C 0.104,E1 3.2684,E2 422.7386} C_DIS
LIN {X 117.8841,Y 68.7548,Z 185,A 32.7296,B 3.1257,C 0.098,E1 3.2653,E2 420.4932} C_DIS
LIN {X 116.2067,Y 71.5538,Z 185,A 33.8735,B 3.1257,C 0.0968,E1 3.2637,E2 419.3772} C_DIS
LIN {X 113.7526,Y 75.3946,Z 185,A 35.598,B 3.1259,C 0.094,E1 3.2611,E2 417.6757} C_DIS
LIN {X 111.6266,Y 78.5074,Z 185,A 37.2373,B 3.1259,C 0.0898,E1 3.2585,E2 416.0288} C_DIS
LIN {X 108.9661,Y 82.1601,Z 185,A 39.053,B 3.1261,C 0.0862,E1 3.2555,E2 414.2227} C_DIS
LIN {X 106.323,Y 85.5531,Z 185,A 40.8166,B 3.1261,C 0.0825,E1 3.2524,E2 412.464} C_DIS
LIN {X 103.5002,Y 88.9473,Z 185,A 42.6063,B 3.1263,C 0.079,E1 3.2492,E2 410.6818} C_DIS
LIN {X 100.5003,Y 92.3232,Z 185,A 44.7805,B 3.1264,C 0.0724,E1 3.2451,E2 408.4728} C_DIS
LIN {X 97.6034,Y 95.381,Z 185,A 45.9616,B 3.1264,C 0.0741,E1 3.2429,E2 407.3642} C_DIS
LIN {X 95.1579,Y 97.8211,Z 185,A 48.1396,B 3.1266,C 0.0646,E1 3.2384,E2 405.0958} C_DIS
LIN {X 91.1151,Y 101.597,Z 185,A 49.5123,B 3.1266,C 0.0685,E1 3.2358,E2 403.8404} C_DIS
LIN {X 88.8067,Y 103.6213,Z 185,A 50.953,B 3.1266,C 0.0647,E1 3.2327,E2 402.381} C_DIS
LIN {X 85.8224,Y 106.1058,Z 185,A 52.6422,B 3.1266,C 0.0612,E1 3.229,E2 400.6845} C_DIS
LIN {X 82.1791,Y 108.9518,Z 185,A 54.5056,B 3.1267,C 0.0584,E1 3.2249,E2 398.8305} C_DIS
LIN {X 78.4107,Y 111.6948,Z 185,A 56.404,B 3.1267,C 0.0555,E1 3.2206,E2 396.9392} C_DIS
LIN {X 74.7828,Y 114.1557,Z 185,A 58.1869,B 3.1268,C 0.053,E1 3.2165,E2 395.1635} C_DIS
LIN {X 71.2025,Y 116.4222,Z 185,A 59.9014,B 3.1268,C 0.0507,E1 3.2124,E2 393.4568} C_DIS
LIN {X 67.4913,Y 118.6121,Z 185,A 61.818,B 3.1269,C 0.0471,E1 3.2078,E2 391.5272} C_DIS
LIN {X 63.0311,Y 121.0398,Z 185,A 63.6919,B 3.1269,C 0.0463,E1 3.2032,E2 389.685} C_DIS
LIN {X 59.9591,Y 122.5906,Z 185,A 65.1032,B 3.1269,C 0.0446,E1 3.1997,E2 388.2779} C_DIS
LIN {X 56.9989,Y 123.9942,Z 185,A 66.4961,B 3.1269,C 0.0427,E1 3.1962,E2 386.883} C_DIS
LIN {X 53.0003,Y 125.7558,Z 185,A 68.4315,B 3.127,C 0.0396,E1 3.1912,E2 384.9356} C_DIS
LIN {X 48.8594,Y 127.4226,Z 185,A 70.3497,B 3.127,C 0.0372,E1 3.1861,E2 383.0124} C_DIS
LIN {X 44.857,Y 128.8846,Z 185,A 71.8538,B 3.127,C 0.0375,E1 3.1823,E2 381.5433} C_DIS
LIN {X 41.4844,Y 130.0093,Z 185,A 73.3239,B 3.127,C 0.0363,E1 3.1784,E2 380.0763} C_DIS
LIN {X 37.7662,Y 131.1391,Z 185,A 74.9073,B 3.127,C 0.0351,E1 3.1742,E2 378.4991} C_DIS
LIN {X 35.0973,Y 131.8771,Z 185,A 76.1,B 3.127,C 0.0339,E1 3.1709,E2 377.303} C_DIS
LIN {X 31.3749,Y 132.8134,Z 185,A 77.7888,B 3.127,C 0.0321,E1 3.1663,E2 375.6053} C_DIS
LIN {X 27.2411,Y 133.7211,Z 185,A 79.4491,B 3.1271,C 0.0317,E1 3.1618,E2 373.9596} C_DIS
LIN {X 23.3183,Y 134.4627,Z 185,A 81.0688,B 3.1271,C 0.0311,E1 3.1574,E2 372.3473} C_DIS
LIN {X 20.053,Y 134.9885,Z 185,A 82.5909,B 3.1271,C 0.0294,E1 3.1531,E2 370.8095} C_DIS
LIN {X 15.7935,Y 135.5513,Z 185,A 84.4616,B 3.1271,C 0.0281,E1 3.1479,E2 368.9313} C_DIS
LIN {X 9.6253,Y 136.1283,Z 185,A 86.5994,B 3.1271,C 0.0304,E1 3.1421,E2 366.8504} C_DIS
LIN {X 6.9493,Y 136.2909,Z 185,A 88.4845,B 3.1271,C 0.0248,E1 3.1366,E2 364.8737} C_DIS
LIN {X 2.4278,Y 136.4465,Z 185,A 89.7601,B 3.1271,C 0.0288,E1 3.1333,E2 363.6746} C_DIS
LIN {X -4.4386,Y 136.3973,Z 185,A 92.6577,B 3.1271,C 0.0284,E1 3.1252,E2 360.7767} C_DIS
LIN {X -10.3155,Y 136.078,Z 185,A 94.995,B 3.1271,C 0.0294,E1 3.1187,E2 358.4567} C_DIS
LIN {X -15.6419,Y 135.5694,Z 185,A 97.3374,B 3.1271,C 0.0292,E1 3.1121,E2 356.1039} C_DIS
LIN {X -19.7266,Y 135.0351,Z 185,A 99.1708,B 3.1271,C 0.0289,E1 3.107,E2 354.2589} C_DIS
LIN {X -23.2925,Y 134.4673,Z 185,A 100.7728,B 3.1271,C 0.0289,E1 3.1026,E2 352.6474} C_DIS
LIN {X -27.1366,Y 133.7424,Z 185,A 102.3721,B 3.1271,C 0.0299,E1 3.0982,E2 351.054} C_DIS
LIN {X -30.7177,Y 132.966,Z 185,A 103.9276,B 3.1271,C 0.0306,E1 3.0939,E2 349.4973} C_DIS
LIN {X -33.8119,Y 132.2128,Z 185,A 105.3044,B 3.1271,C 0.0311,E1 3.0902,E2 348.1165} C_DIS
LIN {X -37.4194,Y 131.2389,Z 185,A 107.1144,B 3.1271,C 0.0307,E1 3.0853,E2 346.2783} C_DIS
LIN {X -41.6053,Y 129.9707,Z 185,A 108.7183,B 3.1271,C 0.0334,E1 3.081,E2 344.7036} C_DIS
LIN {X -44.725,Y 128.9304,Z 185,A 110.1081,B 3.1271,C 0.0344,E1 3.0774,E2 343.3134} C_DIS
LIN {X -48.0293,Y 127.7364,Z 185,A 112.3328,B 3.1271,C 0.0315,E1 3.0713,E2 340.9986} C_DIS
LIN {X -53.1717,Y 125.6842,Z 185,A 113.9567,B 3.1271,C 0.0377,E1 3.0673,E2 339.4615} C_DIS
LIN {X -56.0391,Y 124.4311,Z 185,A 115.2575,B 3.1271,C 0.0391,E1 3.064,E2 338.163} C_DIS
LIN {X -58.7242,Y 123.1861,Z 185,A 116.6497,B 3.1271,C 0.0397,E1 3.0605,E2 336.7535} C_DIS
LIN {X -64.594,Y 120.2145,Z 185,A 119.5613,B 3.127,C 0.0422,E1 3.0532,E2 333.8258} C_DIS
LIN {X -67.4481,Y 118.6368,Z 185,A 120.8961,B 3.127,C 0.0442,E1 3.05,E2 332.4962} C_DIS
LIN {X -72.2254,Y 115.7903,Z 185,A 123.3089,B 3.127,C 0.047,E1 3.0442,E2 330.0755} C_DIS
LIN {X -74.7727,Y 114.1623,Z 185,A 124.5439,B 3.1269,C 0.049,E1 3.0413,E2 328.8456} C_DIS
LIN {X -78.3083,Y 111.7671,Z 185,A 126.4196,B 3.1269,C 0.0513,E1 3.037,E2 326.9612} C_DIS
LIN {X -81.9159,Y 109.1504,Z 185,A 129.0426,B 3.1269,C 0.0507,E1 3.0309,E2 324.2473} C_DIS
LIN {X -86.4977,Y 105.556,Z 185,A 130.5799,B 3.1267,C 0.0592,E1 3.0278,E2 322.823} C_DIS
LIN {X -88.755,Y 103.6658,Z 185,A 132.1388,B 3.1267,C 0.0598,E1 3.0244,E2 321.2258} C_DIS
LIN {X -92.0215,Y 100.7775,Z 185,A 134.0096,B 3.1267,C 0.063,E1 3.0205,E2 319.3514} C_DIS
LIN {X -95.1737,Y 97.8058,Z 185,A 136.08,B 3.1266,C 0.0653,E1 3.0163,E2 317.2516} C_DIS
LIN {X -98.9361,Y 93.9984,Z 185,A 138.2278,B 3.1265,C 0.0701,E1 3.0121,E2 315.1177} C_DIS
LIN {X -101.8902,Y 90.7877,Z 185,A 140.3805,B 3.1265,C 0.0725,E1 3.008,E2 312.927} C_DIS
LIN {X -104.2413,Y 88.078,Z 185,A 142.448,B 3.1265,C 0.0732,E1 3.0042,E2 310.7911} C_DIS
LIN {X -108.1441,Y 83.2402,Z 185,A 144.1335,B 3.1262,C 0.0829,E1 3.0015,E2 309.2217} C_DIS
LIN {X -110.0841,Y 80.6561,Z 185,A 146.9947,B 3.1262,C 0.0795,E1 2.9965,E2 306.1751} C_DIS
LIN {X -114.8455,Y 73.7185,Z 185,A 149.2808,B 3.1259,C 0.0929,E1 2.9932,E2 304.0469} C_DIS
LIN {X -116.7493,Y 70.6646,Z 185,A 150.9626,B 3.1258,C 0.0958,E1 2.9907,E2 302.3453} C_DIS
LIN {X -118.8785,Y 67.0211,Z 185,A 152.8875,B 3.1257,C 0.0995,E1 2.988,E2 300.4028} C_DIS
LIN {X -120.85,Y 63.3925,Z 185,A 154.6421,B 3.1255,C 0.1037,E1 2.9857,E2 298.6469} C_DIS
LIN {X -122.5741,Y 59.9926,Z 185,A 156.269,B 3.1255,C 0.1076,E1 2.9837,E2 297.018} C_DIS
LIN {X -124.6441,Y 55.5628,Z 185,A 158.8182,B 3.1253,C 0.1109,E1 2.9807,E2 294.4087} C_DIS
LIN {X -126.2248,Y 51.8774,Z 185,A 160.1471,B 3.1251,C 0.1166,E1 2.9793,E2 293.1253} C_DIS
LIN {X -127.3996,Y 48.9186,Z 185,A 161.5444,B 3.125,C 0.1199,E1 2.9779,E2 291.7214} C_DIS
LIN {X -129.1262,Y 44.1602,Z 185,A 163.7076,B 3.1248,C 0.1254,E1 2.9758,E2 289.5551} C_DIS
LIN {X -129.9857,Y 41.5584,Z 185,A 165.4481,B 3.1248,C 0.1262,E1 2.9743,E2 287.7418} C_DIS
LIN {X -131.2205,Y 37.4853,Z 185,A 166.8076,B 3.1245,C 0.1326,E1 2.9733,E2 286.4371} C_DIS
LIN {X -132.353,Y 33.2592,Z 185,A 168.8248,B 3.1243,C 0.137,E1 2.9718,E2 284.3987} C_DIS
LIN {X -133.7439,Y 27.1294,Z 185,A 171.4966,B 3.1239,C 0.1441,E1 2.9703,E2 281.7248} C_DIS
LIN {X -134.3581,Y 23.9028,Z 185,A 172.96,B 3.1238,C 0.1476,E1 2.9695,E2 280.2518} C_DIS
LIN {X -134.9378,Y 20.3832,Z 185,A 174.5153,B 3.1236,C 0.1516,E1 2.9688,E2 278.6904} C_DIS
LIN {X -135.4614,Y 16.5472,Z 185,A 176.3101,B 3.1234,C 0.1555,E1 2.9682,E2 276.8754} C_DIS
LIN {X -135.8545,Y 12.9241,Z 185,A 177.8574,B 3.1232,C 0.1597,E1 2.9677,E2 275.327} C_DIS
LIN {X -136.1819,Y 8.8412,Z 185,A 179.7718,B 3.123,C 0.1638,E1 2.9673,E2 273.3892} C_DIS
LIN {X -136.3991,Y 4.3713,Z 185,A -178.2956,B 3.1227,C 0.1689,E1 2.9671,E2 271.4511} C_DIS
LIN {X -136.469,Y 0.3707,Z 185,A -176.4913,B 3.1225,C 0.1732,E1 2.9671,E2 269.6321} C_DIS
LIN {X -136.4152,Y -3.7945,Z 185,A -174.7673,B 3.1222,C 0.1782,E1 2.9671,E2 267.9124} C_DIS
LIN {X -136.2548,Y -7.6581,Z 185,A -172.9513,B 3.122,C 0.182,E1 2.9674,E2 266.073} C_DIS
LIN {X -135.988,Y -11.4339,Z 185,A -171.3924,B 3.1217,C 0.1866,E1 2.9678,E2 264.5189} C_DIS
LIN {X -135.6526,Y -14.8968,Z 185,A -169.8395,B 3.1215,C 0.1903,E1 2.9682,E2 262.9552} C_DIS
LIN {X -135.1288,Y -19.0711,Z 185,A -168.0047,B 3.1212,C 0.195,E1 2.9689,E2 261.1127} C_DIS
LIN {X -134.6042,Y -22.4755,Z 185,A -166.5113,B 3.1209,C 0.1988,E1 2.9696,E2 259.6141} C_DIS
LIN {X -133.9236,Y -26.2352,Z 185,A -164.6979,B 3.1207,C 0.2024,E1 2.9705,E2 257.7748} C_DIS
LIN {X -133.0342,Y -30.4188,Z 185,A -162.9252,B 3.1204,C 0.2074,E1 2.9716,E2 256.006} C_DIS
LIN {X -132.2004,Y -33.8607,Z 185,A -161.3368,B 3.1201,C 0.2111,E1 2.9727,E2 254.4054} C_DIS
LIN {X -131.2946,Y -37.2202,Z 185,A -159.7667,B 3.1199,C 0.2146,E1 2.9739,E2 252.8221} C_DIS
LIN {X -129.0707,Y -44.3203,Z 185,A -156.7793,B 3.1193,C 0.2234,E1 2.9764,E2 249.8539} C_DIS
LIN {X -127.4316,Y -48.8362,Z 185,A -154.5745,B 3.119,C 0.228,E1 2.9785,E2 247.6259} C_DIS
LIN {X -126.3219,Y -51.639,Z 185,A -153.1935,B 3.1187,C 0.2307,E1 2.98,E2 246.2305} C_DIS
LIN {X -124.9342,Y -54.9134,Z 185,A -151.6185,B 3.1185,C 0.2342,E1 2.9817,E2 244.6456} C_DIS
LIN {X -123.4514,Y -58.1689,Z 185,A -149.9429,B 3.1183,C 0.2373,E1 2.9837,E2 242.9481} C_DIS
LIN {X -121.743,Y -61.6608,Z 185,A -148.1406,B 3.118,C 0.2406,E1 2.986,E2 241.1243} C_DIS
LIN {X -119.2483,Y -66.3613,Z 185,A -145.7158,B 3.1176,C 0.2452,E1 2.9893,E2 238.6756} C_DIS
LIN {X -117.6279,Y -69.1923,Z 185,A -144.5168,B 3.1173,C 0.2492,E1 2.991,E2 237.4993} C_DIS
LIN {X -115.2496,Y -73.0856,Z 185,A -142.571,B 3.117,C 0.2535,E1 2.9938,E2 235.5502} C_DIS
LIN {X -112.917,Y -76.6398,Z 185,A -140.6576,B 3.1167,C 0.257,E1 2.9968,E2 233.6206} C_DIS
LIN {X -110.4289,Y -80.1833,Z 185,A -138.7801,B 3.1164,C 0.2608,E1 2.9999,E2 231.7357} C_DIS
LIN {X -107.8486,Y -83.6216,Z 185,A -136.9421,B 3.1161,C 0.2645,E1 3.003,E2 229.8938} C_DIS
LIN {X -105.2248,Y -86.9003,Z 185,A -135.0524,B 3.1158,C 0.2676,E1 3.0064,E2 227.9879} C_DIS
LIN {X -102.3783,Y -90.2364,Z 185,A -133.0645,B 3.1155,C 0.2707,E1 3.01,E2 225.9812} C_DIS
LIN {X -98.7342,Y -94.2097,Z 185,A -130.9986,B 3.1151,C 0.2761,E1 3.0139,E2 223.9416} C_DIS
LIN {X -96.0847,Y -96.9105,Z 185,A -129.3354,B 3.1148,C 0.2788,E1 3.0172,E2 222.2688} C_DIS
LIN {X -93.3462,Y -99.5517,Z 185,A -127.5483,B 3.1146,C 0.2808,E1 3.0209,E2 220.457} C_DIS
LIN {X -90.0597,Y -102.5346,Z 185,A -125.6172,B 3.1144,C 0.2837,E1 3.0249,E2 218.5172} C_DIS
LIN {X -86.6775,Y -105.409,Z 185,A -123.6941,B 3.1141,C 0.2866,E1 3.0291,E2 216.5864} C_DIS
LIN {X -83.2458,Y -108.1398,Z 185,A -121.8011,B 3.1139,C 0.2893,E1 3.0333,E2 214.6867} C_DIS
LIN {X -79.6811,Y -110.7924,Z 185,A -119.8586,B 3.1136,C 0.2917,E1 3.0377,E2 212.734} C_DIS
LIN {X -75.8174,Y -113.4708,Z 185,A -117.9438,B 3.1133,C 0.295,E1 3.0421,E2 210.827} C_DIS
LIN {X -72.2856,Y -115.7529,Z 185,A -116.0666,B 3.1132,C 0.2968,E1 3.0465,E2 208.9349} C_DIS
LIN {X -67.9275,Y -118.3633,Z 185,A -114.0141,B 3.1129,C 0.3,E1 3.0515,E2 206.8929} C_DIS
LIN {X -64.6441,Y -120.1875,Z 185,A -112.3205,B 3.1127,C 0.3012,E1 3.0556,E2 205.1837} C_DIS
LIN {X -61.5939,Y -121.777,Z 185,A -110.9114,B 3.1126,C 0.3031,E1 3.0591,E2 203.7791} C_DIS
LIN {X -58.095,Y -123.4867,Z 185,A -109.246,B 3.1124,C 0.3047,E1 3.0634,E2 202.1095} C_DIS
LIN {X -55.1527,Y -124.8275,Z 185,A -107.7091,B 3.1124,C 0.3049,E1 3.0673,E2 200.5485} C_DIS
LIN {X -51.7799,Y -126.2651,Z 185,A -106.0171,B 3.1124,C 0.3054,E1 3.0718,E2 198.836} C_DIS
LIN {X -47.8108,Y -127.8182,Z 185,A -104.4829,B 3.112,C 0.3085,E1 3.0757,E2 197.3353} C_DIS
LIN {X -44.5214,Y -129.001,Z 185,A -103.0614,B 3.1119,C 0.31,E1 3.0794,E2 195.9196} C_DIS
LIN {X -41.4986,Y -130.0048,Z 185,A -101.6133,B 3.1119,C 0.3102,E1 3.0833,E2 194.4565} C_DIS
LIN {X -37.4446,Y -131.2319,Z 185,A -99.7271,B 3.1119,C 0.3107,E1 3.0884,E2 192.5554} C_DIS
LIN {X -33.605,Y -132.2653,Z 185,A -98.166,B 3.1116,C 0.3123,E1 3.0926,E2 191.0082} C_DIS
LIN {X -30.0135,Y -133.1268,Z 185,A -96.6267,B 3.1116,C 0.3131,E1 3.0968,E2 189.4699} C_DIS
LIN {X -26.5294,Y -133.866,Z 185,A -95.1154,B 3.1116,C 0.3136,E1 3.1009,E2 187.9561} C_DIS
LIN {X -23.5302,Y -134.4248,Z 185,A -93.7581,B 3.1116,C 0.3136,E1 3.1047,E2 186.5882} C_DIS
LIN {X -19.3973,Y -135.0822,Z 185,A -91.0141,B 3.1122,C 0.307,E1 3.1127,E2 183.711} C_DIS
LIN {X -12.1419,Y -135.9282,Z 185,A -88.1427,B 3.112,C 0.3087,E1 3.1206,E2 180.8648} C_DIS
LIN {X -5.9856,Y -136.3382,Z 185,A -86.4466,B 3.1114,C 0.3152,E1 3.125,E2 179.2876} C_DIS
LIN {X -0.0569,Y -136.4697,Z 185,A -83.9273,B 3.1114,C 0.3146,E1 3.132,E2 176.7634} C_DIS
LIN {X -0.0569,Y -136.4697,Z 185,A -83.9274,B 3.1114,C 0.3146,E1 3.132,E2 176.7634} C_DIS
Enddeposition()
LIN {X 0.9714,Y -137.3619,Z 185,A -83.6425,B 3.1206,C 0.3176,E1 3.1421,E2 176.5256} C_DIS
Startdeposition()
$VEL.CP = VEL_PRINT
LIN {X -1.8733,Y -137.356,Z 185,A -85.3262,B 3.1202,C 0.3215,E1 3.1372,E2 178.2763} C_DIS
LIN {X -5.7119,Y -137.2497,Z 185,A -87.0636,B 3.12,C 0.3226,E1 3.1323,E2 180.0325} C_DIS
LIN {X -11.8774,Y -136.8539,Z 185,A -89.522,B 3.1201,C 0.3216,E1 3.1255,E2 182.4763} C_DIS
LIN {X -16.2133,Y -136.4078,Z 185,A -91.3439,B 3.1201,C 0.3214,E1 3.1204,E2 184.2993} C_DIS
LIN {X -19.7026,Y -135.9479,Z 185,A -93.1252,B 3.12,C 0.3232,E1 3.1154,E2 186.1227} C_DIS
LIN {X -23.56,Y -135.334,Z 185,A -94.4917,B 3.1202,C 0.3209,E1 3.1117,E2 187.4551} C_DIS
LIN {X -27.249,Y -134.6382,Z 185,A -95.9949,B 3.1203,C 0.3199,E1 3.1076,E2 188.9504} C_DIS
LIN {X -31.1384,Y -133.7932,Z 185,A -97.645,B 3.1204,C 0.3191,E1 3.1031,E2 190.5997} C_DIS
LIN {X -34.9731,Y -132.8419,Z 185,A -99.3318,B 3.1204,C 0.3185,E1 3.0985,E2 192.2922} C_DIS
LIN {X -38.3823,Y -131.8967,Z 185,A -100.746,B 3.1206,C 0.3172,E1 3.0947,E2 193.6987} C_DIS
LIN {X -41.507,Y -130.9471,Z 185,A -102.1308,B 3.1206,C 0.3164,E1 3.091,E2 195.0868} C_DIS
LIN {X -44.3935,Y -129.9981,Z 185,A -103.3516,B 3.1208,C 0.3152,E1 3.0878,E2 196.3017} C_DIS
LIN {X -47.8055,Y -128.7815,Z 185,A -104.8437,B 3.1209,C 0.3138,E1 3.0839,E2 197.7916} C_DIS
LIN {X -51.3649,Y -127.4029,Z 185,A -106.4196,B 3.1211,C 0.3124,E1 3.0798,E2 199.3658} C_DIS
LIN {X -54.4022,Y -126.1359,Z 185,A -108.004,B 3.1211,C 0.3124,E1 3.0756,E2 200.9784} C_DIS
LIN {X -57.5477,Y -124.7322,Z 185,A -109.4305,B 3.1212,C 0.3108,E1 3.072,E2 202.4038} C_DIS
LIN {X -60.726,Y -123.2161,Z 185,A -110.9741,B 3.1214,C 0.3097,E1 3.0681,E2 203.9575} C_DIS
LIN {X -63.724,Y -121.6927,Z 185,A -112.3475,B 3.1215,C 0.3079,E1 3.0647,E2 205.3272} C_DIS
LIN {X -67.5113,Y -119.6356,Z 185,A -114.2041,B 3.1217,C 0.306,E1 3.0601,E2 207.1919} C_DIS
LIN {X -70.9275,Y -117.6424,Z 185,A -115.982,B 3.1219,C 0.3046,E1 3.0558,E2 208.9867} C_DIS
LIN {X -74.8479,Y -115.1876,Z 185,A -117.931,B 3.1221,C 0.302,E1 3.0512,E2 210.9384} C_DIS
LIN {X -78.5225,Y -112.7148,Z 185,A -119.8341,B 3.1223,C 0.2996,E1 3.0468,E2 212.8489} C_DIS
LIN {X -82.0747,Y -110.1551,Z 185,A -121.7138,B 3.1226,C 0.2971,E1 3.0426,E2 214.7355} C_DIS
LIN {X -85.6795,Y -107.3753,Z 185,A -123.6444,B 3.1229,C 0.2942,E1 3.0383,E2 216.6702} C_DIS
LIN {X -89.2081,Y -104.4624,Z 185,A -125.6414,B 3.1231,C 0.2914,E1 3.034,E2 218.6787} C_DIS
LIN {X -92.6407,Y -101.4312,Z 185,A -127.6282,B 3.1234,C 0.2884,E1 3.0299,E2 220.6754} C_DIS
LIN {X -96.1545,Y -98.1056,Z 185,A -129.9768,B 3.1236,C 0.2863,E1 3.0251,E2 223.0668} C_DIS
LIN {X -98.8368,Y -95.4029,Z 185,A -132.171,B 3.1236,C 0.2862,E1 3.0207,E2 225.3392} C_DIS
LIN {X -103.365,Y -90.4772,Z 185,A -134.203,B 3.1244,C 0.2769,E1 3.0171,E2 227.2725} C_DIS
LIN {X -106.2102,Y -87.1198,Z 185,A -136.0939,B 3.1247,C 0.2733,E1 3.0137,E2 229.1702} C_DIS
LIN {X -108.8373,Y -83.8154,Z 185,A -137.9323,B 3.125,C 0.2699,E1 3.0105,E2 231.0183} C_DIS
LIN {X -111.4211,Y -80.3483,Z 185,A -139.8069,B 3.1254,C 0.2663,E1 3.0074,E2 232.9017} C_DIS
LIN {X -113.9766,Y -76.6803,Z 185,A -141.7512,B 3.1257,C 0.2624,E1 3.0043,E2 234.8558} C_DIS
LIN {X -116.4089,Y -72.9352,Z 185,A -143.7142,B 3.126,C 0.2586,E1 3.0013,E2 236.8311} C_DIS
LIN {X -118.4235,Y -69.6152,Z 185,A -145.3025,B 3.1263,C 0.2546,E1 2.9991,E2 238.4149} C_DIS
LIN {X -120.5092,Y -65.9392,Z 185,A -147.199,B 3.1266,C 0.2509,E1 2.9965,E2 240.328} C_DIS
LIN {X -122.4759,Y -62.2054,Z 185,A -148.9422,B 3.127,C 0.2465,E1 2.9942,E2 242.0683} C_DIS
LIN {X -124.046,Y -59.0125,Z 185,A -150.5019,B 3.1272,C 0.2431,E1 2.9923,E2 243.6372} C_DIS
LIN {X -125.882,Y -54.9895,Z 185,A -152.4506,B 3.1276,C 0.2389,E1 2.9901,E2 245.5986} C_DIS
Enddeposition()
END
